Yaskawa INFORM job: A_ROOF_UPPER_0614_2_PAINT_1.JBI

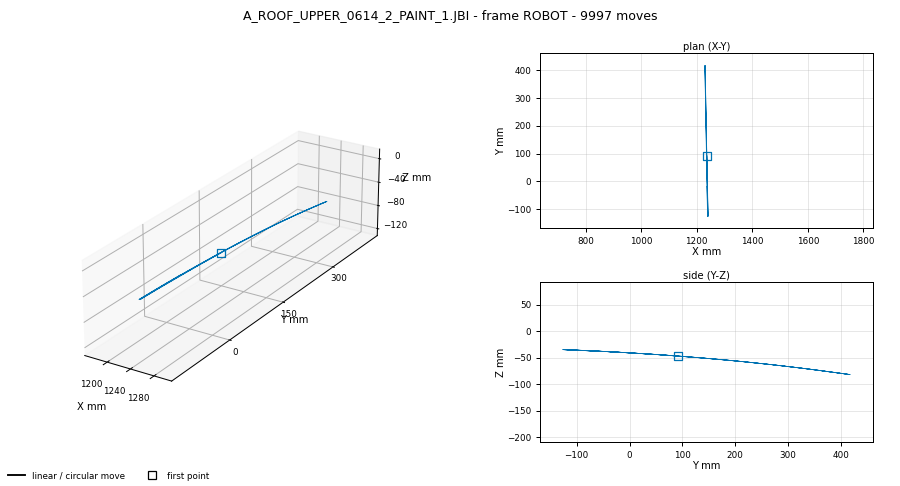
[picture p0: tool path of A_ROOF_UPPER_0614_2_PAINT_1.JBI in frame ROBOT, 9997 of 9997 moves have a stored position in this frame; points joined in program order, loops and branches not executed]
/JOB
//NAME A_ROOF_UPPER_0614_2_PAINT1
//POS
///NPOS 9997,0,0,0,0,0
///TOOL 1
///USER 0
///POSTYPE ROBOT
///RECTAN
///RCONF 1,0,0,0,0,0,0,0,0,0,0,0,0,0,0,0,0,0,0,0,0,0,0,0
C00000=1236.854,92.154,-46.600,-178.429,5.415,148.469
C00001=1236.860,91.904,-46.581,-178.431,5.414,148.469
C00002=1236.864,91.655,-46.563,-178.434,5.413,148.470
C00003=1236.868,91.406,-46.544,-178.436,5.413,148.471
C00004=1236.874,91.156,-46.525,-178.439,5.412,148.471
C00005=1236.879,90.907,-46.507,-178.441,5.411,148.472
C00006=1236.884,90.658,-46.489,-178.444,5.411,148.472
C00007=1236.888,90.409,-46.470,-178.446,5.410,148.473
C00008=1236.894,90.159,-46.452,-178.449,5.409,148.474
C00009=1236.898,89.911,-46.433,-178.452,5.409,148.474
C00010=1236.903,89.661,-46.415,-178.454,5.408,148.475
C00011=1236.907,89.411,-46.397,-178.456,5.407,148.476
C00012=1236.913,89.162,-46.378,-178.459,5.407,148.476
C00013=1236.918,88.913,-46.359,-178.462,5.406,148.477
C00014=1236.922,88.664,-46.341,-178.464,5.405,148.477
C00015=1236.927,88.414,-46.323,-178.467,5.404,148.478
C00016=1236.932,88.165,-46.305,-178.470,5.403,148.479
C00017=1236.937,87.916,-46.286,-178.472,5.402,148.479
C00018=1236.941,87.666,-46.268,-178.475,5.402,148.480
C00019=1236.946,87.417,-46.250,-178.477,5.401,148.480
C00020=1236.951,87.168,-46.232,-178.480,5.400,148.481
C00021=1236.956,86.919,-46.214,-178.482,5.400,148.482
C00022=1236.961,86.669,-46.195,-178.485,5.399,148.482
C00023=1236.966,86.420,-46.176,-178.487,5.398,148.483
C00024=1236.971,86.171,-46.158,-178.490,5.397,148.483
C00025=1236.976,85.922,-46.140,-178.492,5.397,148.484
C00026=1236.980,85.672,-46.122,-178.495,5.396,148.485
C00027=1236.985,85.423,-46.104,-178.497,5.396,148.485
C00028=1236.990,85.174,-46.086,-178.500,5.395,148.486
C00029=1236.995,84.924,-46.067,-178.502,5.394,148.486
C00030=1237.000,84.676,-46.048,-178.505,5.393,148.487
C00031=1237.004,84.426,-46.030,-178.507,5.393,148.488
C00032=1237.009,84.176,-46.012,-178.510,5.392,148.488
C00033=1237.014,83.927,-45.994,-178.513,5.392,148.489
C00034=1237.019,83.678,-45.976,-178.515,5.391,148.489
C00035=1237.024,83.429,-45.958,-178.517,5.390,148.490
C00036=1237.029,83.180,-45.940,-178.520,5.389,148.491
C00037=1237.033,82.930,-45.922,-178.523,5.389,148.491
C00038=1237.038,82.681,-45.904,-178.525,5.388,148.492
C00039=1237.043,82.432,-45.886,-178.527,5.387,148.492
C00040=1237.049,82.163,-45.866,-178.530,5.387,148.493
C00041=1237.054,81.895,-45.846,-178.533,5.386,148.494
C00042=1237.059,81.626,-45.827,-178.536,5.385,148.494
C00043=1237.064,81.358,-45.808,-178.539,5.384,148.495
C00044=1237.069,81.109,-45.790,-178.541,5.383,148.496
C00045=1237.074,80.860,-45.772,-178.544,5.383,148.496
C00046=1237.078,80.610,-45.753,-178.546,5.382,148.497
C00047=1237.083,80.361,-45.735,-178.549,5.382,148.498
C00048=1237.088,80.112,-45.717,-178.552,5.381,148.498
C00049=1237.093,79.862,-45.699,-178.554,5.380,148.499
C00050=1237.098,79.613,-45.682,-178.556,5.379,148.499
C00051=1237.103,79.364,-45.664,-178.559,5.379,148.500
C00052=1237.108,79.114,-45.646,-178.562,5.378,148.501
C00053=1237.113,78.865,-45.628,-178.564,5.378,148.501
C00054=1237.117,78.615,-45.610,-178.566,5.377,148.502
C00055=1237.122,78.366,-45.592,-178.569,5.376,148.502
C00056=1237.127,78.117,-45.574,-178.572,5.375,148.503
C00057=1237.132,77.868,-45.556,-178.574,5.375,148.504
C00058=1237.137,77.619,-45.538,-178.577,5.374,148.504
C00059=1237.142,77.369,-45.520,-178.580,5.374,148.505
C00060=1237.147,77.120,-45.503,-178.582,5.373,148.506
C00061=1237.152,76.870,-45.485,-178.584,5.372,148.506
C00062=1237.157,76.621,-45.467,-178.587,5.371,148.507
C00063=1237.162,76.372,-45.449,-178.590,5.371,148.508
C00064=1237.167,76.123,-45.431,-178.592,5.370,148.508
C00065=1237.172,75.873,-45.414,-178.595,5.370,148.509
C00066=1237.176,75.623,-45.395,-178.597,5.369,148.509
C00067=1237.180,75.374,-45.378,-178.600,5.368,148.510
C00068=1237.185,75.125,-45.360,-178.602,5.368,148.511
C00069=1237.190,74.876,-45.342,-178.605,5.367,148.511
C00070=1237.195,74.626,-45.325,-178.607,5.367,148.512
C00071=1237.200,74.377,-45.307,-178.610,5.367,148.513
C00072=1237.205,74.128,-45.289,-178.612,5.366,148.513
C00073=1237.210,73.879,-45.271,-178.614,5.365,148.514
C00074=1237.215,73.629,-45.253,-178.617,5.364,148.514
C00075=1237.220,73.380,-45.236,-178.620,5.364,148.515
C00076=1237.224,73.131,-45.218,-178.622,5.363,148.516
C00077=1237.230,72.881,-45.201,-178.625,5.363,148.516
C00078=1237.235,72.632,-45.183,-178.627,5.362,148.517
C00079=1237.240,72.383,-45.165,-178.630,5.361,148.517
C00080=1237.244,72.134,-45.147,-178.632,5.360,148.518
C00081=1237.249,71.884,-45.130,-178.635,5.360,148.519
C00082=1237.254,71.635,-45.112,-178.637,5.359,148.519
C00083=1237.259,71.386,-45.094,-178.640,5.359,148.520
C00084=1237.264,71.136,-45.077,-178.643,5.358,148.521
C00085=1237.269,70.887,-45.059,-178.645,5.357,148.521
C00086=1237.273,70.637,-45.042,-178.647,5.357,148.522
C00087=1237.278,70.388,-45.024,-178.650,5.356,148.522
C00088=1237.283,70.139,-45.006,-178.653,5.355,148.523
C00089=1237.288,69.889,-44.989,-178.655,5.355,148.524
C00090=1237.293,69.640,-44.972,-178.658,5.354,148.524
C00091=1237.298,69.390,-44.954,-178.661,5.354,148.525
C00092=1237.303,69.141,-44.936,-178.663,5.353,148.526
C00093=1237.308,68.892,-44.918,-178.666,5.352,148.526
C00094=1237.312,68.643,-44.902,-178.668,5.351,148.527
C00095=1237.317,68.393,-44.884,-178.670,5.352,148.528
C00096=1237.322,68.144,-44.866,-178.673,5.351,148.528
C00097=1237.327,67.894,-44.849,-178.675,5.350,148.529
C00098=1237.332,67.645,-44.832,-178.678,5.350,148.530
C00099=1237.337,67.396,-44.814,-178.681,5.349,148.530
C00100=1237.342,67.146,-44.797,-178.683,5.349,148.531
C00101=1237.346,66.897,-44.779,-178.685,5.348,148.531
C00102=1237.352,66.648,-44.762,-178.688,5.347,148.532
C00103=1237.357,66.399,-44.744,-178.691,5.347,148.533
C00104=1237.362,66.149,-44.727,-178.693,5.346,148.533
C00105=1237.366,65.900,-44.710,-178.696,5.345,148.534
C00106=1237.371,65.650,-44.692,-178.699,5.345,148.535
C00107=1237.376,65.401,-44.674,-178.701,5.344,148.535
C00108=1237.381,65.152,-44.658,-178.704,5.344,148.536
C00109=1237.386,64.903,-44.640,-178.706,5.343,148.536
C00110=1237.391,64.653,-44.623,-178.708,5.343,148.537
C00111=1237.395,64.403,-44.606,-178.711,5.342,148.538
C00112=1237.400,64.154,-44.588,-178.713,5.342,148.538
C00113=1237.405,63.905,-44.572,-178.716,5.341,148.539
C00114=1237.410,63.656,-44.554,-178.719,5.340,148.540
C00115=1237.415,63.406,-44.536,-178.721,5.340,148.540
C00116=1237.420,63.157,-44.520,-178.724,5.339,148.541
C00117=1237.425,62.908,-44.502,-178.726,5.339,148.542
C00118=1237.429,62.658,-44.485,-178.729,5.338,148.542
C00119=1237.434,62.409,-44.467,-178.731,5.337,148.543
C00120=1237.439,62.159,-44.450,-178.734,5.337,148.543
C00121=1237.444,61.910,-44.433,-178.736,5.336,148.544
C00122=1237.449,61.661,-44.415,-178.739,5.335,148.545
C00123=1237.454,61.412,-44.399,-178.741,5.336,148.545
C00124=1237.459,61.162,-44.382,-178.744,5.335,148.546
C00125=1237.464,60.912,-44.364,-178.746,5.334,148.547
C00126=1237.468,60.663,-44.347,-178.749,5.334,148.547
C00127=1237.474,60.414,-44.330,-178.752,5.333,148.548
C00128=1237.479,60.165,-44.313,-178.754,5.332,148.549
C00129=1237.484,59.916,-44.295,-178.756,5.332,148.549
C00130=1237.488,59.666,-44.279,-178.759,5.331,148.550
C00131=1237.493,59.416,-44.261,-178.762,5.331,148.551
C00132=1237.498,59.167,-44.245,-178.764,5.330,148.551
C00133=1237.503,58.918,-44.227,-178.767,5.329,148.552
C00134=1237.508,58.669,-44.210,-178.769,5.330,148.553
C00135=1237.513,58.419,-44.193,-178.772,5.329,148.553
C00136=1237.518,58.170,-44.177,-178.774,5.328,148.554
C00137=1237.523,57.920,-44.159,-178.777,5.328,148.555
C00138=1237.528,57.672,-44.142,-178.779,5.327,148.555
C00139=1237.533,57.422,-44.125,-178.782,5.326,148.556
C00140=1237.537,57.172,-44.108,-178.784,5.326,148.556
C00141=1237.542,56.923,-44.091,-178.787,5.325,148.557
C00142=1237.547,56.673,-44.074,-178.790,5.325,148.558
C00143=1237.553,56.424,-44.057,-178.792,5.325,148.558
C00144=1237.557,56.155,-44.039,-178.795,5.323,148.559
C00145=1237.563,55.887,-44.021,-178.798,5.323,148.560
C00146=1237.568,55.619,-44.003,-178.800,5.322,148.560
C00147=1237.573,55.350,-43.984,-178.803,5.322,148.561
C00148=1237.578,55.102,-43.967,-178.805,5.322,148.562
C00149=1237.583,54.852,-43.950,-178.808,5.321,148.562
C00150=1237.588,54.602,-43.933,-178.810,5.321,148.563
C00151=1237.592,54.353,-43.917,-178.813,5.320,148.564
C00152=1237.598,54.104,-43.900,-178.815,5.320,148.564
C00153=1237.603,53.854,-43.883,-178.818,5.319,148.565
C00154=1237.608,53.605,-43.866,-178.821,5.318,148.566
C00155=1237.612,53.355,-43.849,-178.823,5.318,148.566
C00156=1237.617,53.106,-43.833,-178.826,5.317,148.567
C00157=1237.623,52.856,-43.816,-178.828,5.317,148.568
C00158=1237.627,52.607,-43.799,-178.831,5.317,148.568
C00159=1237.633,52.358,-43.782,-178.833,5.316,148.569
C00160=1237.637,52.108,-43.765,-178.836,5.316,148.570
C00161=1237.642,51.859,-43.749,-178.838,5.315,148.570
C00162=1237.647,51.609,-43.731,-178.841,5.314,148.571
C00163=1237.652,51.360,-43.715,-178.843,5.314,148.571
C00164=1237.657,51.111,-43.698,-178.846,5.313,148.572
C00165=1237.662,50.861,-43.681,-178.848,5.313,148.573
C00166=1237.667,50.612,-43.665,-178.851,5.313,148.574
C00167=1237.672,50.363,-43.648,-178.853,5.312,148.574
C00168=1237.676,50.113,-43.632,-178.856,5.312,148.575
C00169=1237.682,49.864,-43.615,-178.859,5.311,148.576
C00170=1237.686,49.615,-43.598,-178.861,5.310,148.576
C00171=1237.691,49.365,-43.581,-178.864,5.310,148.577
C00172=1237.697,49.116,-43.564,-178.866,5.310,148.578
C00173=1237.701,48.867,-43.548,-178.869,5.309,148.578
C00174=1237.706,48.617,-43.531,-178.871,5.309,148.579
C00175=1237.712,48.367,-43.515,-178.874,5.308,148.580
C00176=1237.716,48.118,-43.498,-178.876,5.307,148.580
C00177=1237.721,47.868,-43.482,-178.879,5.307,148.581
C00178=1237.726,47.620,-43.465,-178.881,5.306,148.581
C00179=1237.731,47.370,-43.448,-178.883,5.306,148.582
C00180=1237.735,47.120,-43.431,-178.886,5.306,148.583
C00181=1237.740,46.872,-43.415,-178.889,5.305,148.583
C00182=1237.745,46.622,-43.399,-178.891,5.305,148.584
C00183=1237.750,46.372,-43.382,-178.894,5.304,148.585
C00184=1237.756,46.123,-43.365,-178.897,5.304,148.585
C00185=1237.760,45.873,-43.349,-178.899,5.303,148.586
C00186=1237.765,45.625,-43.333,-178.901,5.303,148.587
C00187=1237.770,45.375,-43.317,-178.904,5.303,148.587
C00188=1237.775,45.125,-43.299,-178.907,5.302,148.588
C00189=1237.780,44.876,-43.283,-178.909,5.301,148.589
C00190=1237.785,44.627,-43.266,-178.912,5.301,148.589
C00191=1237.790,44.378,-43.250,-178.914,5.300,148.590
C00192=1237.795,44.128,-43.234,-178.917,5.301,148.591
C00193=1237.799,43.878,-43.217,-178.919,5.300,148.591
C00194=1237.805,43.629,-43.200,-178.922,5.299,148.592
C00195=1237.810,43.379,-43.185,-178.924,5.299,148.593
C00196=1237.815,43.130,-43.168,-178.927,5.298,148.593
C00197=1237.819,42.881,-43.152,-178.929,5.297,148.594
C00198=1237.824,42.631,-43.135,-178.931,5.298,148.595
C00199=1237.829,42.382,-43.119,-178.934,5.297,148.595
C00200=1237.834,42.132,-43.102,-178.937,5.296,148.596
C00201=1237.839,41.883,-43.086,-178.939,5.296,148.597
C00202=1237.844,41.633,-43.070,-178.942,5.295,148.597
C00203=1237.849,41.384,-43.053,-178.944,5.295,148.598
C00204=1237.854,41.135,-43.037,-178.947,5.295,148.599
C00205=1237.859,40.885,-43.021,-178.949,5.294,148.599
C00206=1237.864,40.636,-43.005,-178.952,5.294,148.600
C00207=1237.868,40.387,-42.988,-178.954,5.293,148.601
C00208=1237.873,40.137,-42.972,-178.957,5.293,148.601
C00209=1237.878,39.888,-42.956,-178.960,5.292,148.602
C00210=1237.884,39.638,-42.939,-178.962,5.292,148.603
C00211=1237.889,39.388,-42.923,-178.964,5.292,148.603
C00212=1237.894,39.140,-42.906,-178.967,5.291,148.604
C00213=1237.898,38.890,-42.891,-178.970,5.291,148.605
C00214=1237.903,38.641,-42.874,-178.972,5.290,148.605
C00215=1237.908,38.391,-42.858,-178.974,5.290,148.606
C00216=1237.913,38.142,-42.842,-178.977,5.290,148.607
C00217=1237.918,37.892,-42.826,-178.980,5.289,148.607
C00218=1237.923,37.643,-42.810,-178.982,5.289,148.608
C00219=1237.928,37.393,-42.794,-178.985,5.288,148.609
C00220=1237.933,37.144,-42.777,-178.987,5.288,148.609
C00221=1237.938,36.895,-42.761,-178.990,5.288,148.610
C00222=1237.943,36.645,-42.745,-178.992,5.287,148.611
C00223=1237.947,36.396,-42.729,-178.995,5.287,148.611
C00224=1237.953,36.146,-42.713,-178.998,5.286,148.612
C00225=1237.957,35.897,-42.696,-179.000,5.285,148.613
C00226=1237.963,35.647,-42.681,-179.002,5.285,148.613
C00227=1237.967,35.397,-42.665,-179.005,5.285,148.614
C00228=1237.973,35.149,-42.648,-179.007,5.284,148.615
C00229=1237.978,34.899,-42.633,-179.010,5.284,148.615
C00230=1237.982,34.650,-42.616,-179.012,5.283,148.616
C00231=1237.988,34.400,-42.601,-179.014,5.283,148.617
C00232=1237.992,34.151,-42.584,-179.017,5.283,148.617
C00233=1237.998,33.901,-42.568,-179.020,5.282,148.618
C00234=1238.002,33.652,-42.552,-179.022,5.282,148.619
C00235=1238.008,33.402,-42.536,-179.025,5.281,148.619
C00236=1238.012,33.152,-42.520,-179.027,5.281,148.620
C00237=1238.017,32.904,-42.504,-179.030,5.281,148.621
C00238=1238.022,32.655,-42.489,-179.032,5.280,148.621
C00239=1238.027,32.404,-42.473,-179.035,5.280,148.622
C00240=1238.032,32.156,-42.457,-179.038,5.279,148.623
C00241=1238.037,31.906,-42.441,-179.040,5.279,148.623
C00242=1238.042,31.657,-42.424,-179.042,5.279,148.624
C00243=1238.047,31.407,-42.408,-179.045,5.278,148.625
C00244=1238.052,31.157,-42.393,-179.048,5.278,148.625
C00245=1238.057,30.908,-42.376,-179.050,5.278,148.626
C00246=1238.062,30.658,-42.360,-179.052,5.277,148.627
C00247=1238.066,30.409,-42.345,-179.055,5.277,148.627
C00248=1238.072,30.141,-42.328,-179.058,5.276,148.628
C00249=1238.077,29.872,-42.311,-179.061,5.276,148.629
C00250=1238.083,29.603,-42.294,-179.064,5.275,148.630
C00251=1238.088,29.335,-42.277,-179.066,5.275,148.630
C00252=1238.093,29.086,-42.261,-179.068,5.275,148.631
C00253=1238.098,28.836,-42.245,-179.071,5.275,148.632
C00254=1238.103,28.587,-42.230,-179.074,5.274,148.632
C00255=1238.108,28.337,-42.214,-179.076,5.273,148.633
C00256=1238.112,28.088,-42.198,-179.079,5.273,148.634
C00257=1238.118,27.838,-42.182,-179.081,5.273,148.635
C00258=1238.123,27.588,-42.166,-179.084,5.273,148.635
C00259=1238.128,27.339,-42.150,-179.086,5.272,148.636
C00260=1238.133,27.090,-42.135,-179.089,5.271,148.637
C00261=1238.137,26.840,-42.119,-179.091,5.272,148.637
C00262=1238.143,26.591,-42.103,-179.094,5.271,148.638
C00263=1238.148,26.341,-42.088,-179.096,5.271,148.639
C00264=1238.152,26.092,-42.072,-179.099,5.270,148.639
C00265=1238.157,25.842,-42.057,-179.101,5.269,148.640
C00266=1238.163,25.593,-42.041,-179.104,5.270,148.641
C00267=1238.167,25.343,-42.024,-179.106,5.269,148.641
C00268=1238.172,25.094,-42.009,-179.109,5.269,148.642
C00269=1238.177,24.845,-41.994,-179.111,5.268,148.643
C00270=1238.182,24.595,-41.978,-179.114,5.268,148.643
C00271=1238.187,24.345,-41.962,-179.116,5.268,148.644
C00272=1238.192,24.096,-41.947,-179.119,5.267,148.645
C00273=1238.198,23.847,-41.932,-179.121,5.267,148.645
C00274=1238.202,23.597,-41.916,-179.124,5.267,148.646
C00275=1238.207,23.348,-41.899,-179.126,5.266,148.647
C00276=1238.212,23.099,-41.884,-179.129,5.266,148.647
C00277=1238.217,22.849,-41.868,-179.131,5.265,148.648
C00278=1238.222,22.599,-41.853,-179.134,5.265,148.649
C00279=1238.227,22.350,-41.838,-179.136,5.265,148.649
C00280=1238.232,22.101,-41.822,-179.139,5.264,148.650
C00281=1238.237,21.851,-41.806,-179.142,5.264,148.651
C00282=1238.242,21.602,-41.791,-179.144,5.264,148.652
C00283=1238.247,21.352,-41.776,-179.146,5.264,148.652
C00284=1238.252,21.102,-41.760,-179.149,5.263,148.653
C00285=1238.256,20.853,-41.745,-179.152,5.262,148.654
C00286=1238.262,20.604,-41.729,-179.154,5.263,148.654
C00287=1238.267,20.354,-41.714,-179.156,5.262,148.655
C00288=1238.271,20.105,-41.698,-179.159,5.262,148.656
C00289=1238.277,19.855,-41.683,-179.162,5.261,148.656
C00290=1238.282,19.606,-41.667,-179.164,5.261,148.657
C00291=1238.287,19.357,-41.652,-179.166,5.261,148.658
C00292=1238.292,19.107,-41.637,-179.169,5.260,148.658
C00293=1238.296,18.857,-41.621,-179.172,5.260,148.659
C00294=1238.302,18.608,-41.606,-179.174,5.260,148.660
C00295=1238.307,18.359,-41.590,-179.177,5.260,148.661
C00296=1238.312,18.110,-41.575,-179.179,5.259,148.661
C00297=1238.317,17.859,-41.560,-179.182,5.259,148.662
C00298=1238.321,17.610,-41.545,-179.184,5.259,148.663
C00299=1238.327,17.360,-41.529,-179.187,5.258,148.663
C00300=1238.331,17.111,-41.514,-179.189,5.258,148.664
C00301=1238.337,16.862,-41.499,-179.192,5.257,148.665
C00302=1238.342,16.612,-41.483,-179.194,5.257,148.665
C00303=1238.346,16.363,-41.468,-179.197,5.257,148.666
C00304=1238.352,16.113,-41.452,-179.199,5.256,148.667
C00305=1238.357,15.864,-41.438,-179.202,5.257,148.667
C00306=1238.362,15.614,-41.422,-179.204,5.256,148.668
C00307=1238.366,15.364,-41.407,-179.207,5.256,148.669
C00308=1238.371,15.115,-41.391,-179.209,5.255,148.670
C00309=1238.376,14.866,-41.376,-179.212,5.255,148.670
C00310=1238.381,14.616,-41.361,-179.214,5.255,148.671
C00311=1238.386,14.367,-41.346,-179.217,5.254,148.672
C00312=1238.392,14.117,-41.331,-179.219,5.254,148.672
C00313=1238.396,13.868,-41.316,-179.222,5.254,148.673
C00314=1238.401,13.618,-41.300,-179.224,5.253,148.674
C00315=1238.406,13.369,-41.285,-179.227,5.253,148.674
C00316=1238.412,13.119,-41.270,-179.229,5.253,148.675
C00317=1238.416,12.870,-41.255,-179.232,5.252,148.676
C00318=1238.422,12.621,-41.239,-179.234,5.252,148.676
C00319=1238.426,12.371,-41.224,-179.237,5.251,148.677
C00320=1238.432,12.121,-41.210,-179.239,5.252,148.678
C00321=1238.436,11.872,-41.194,-179.242,5.251,148.678
C00322=1238.441,11.622,-41.179,-179.244,5.251,148.679
C00323=1238.446,11.372,-41.164,-179.246,5.251,148.680
C00324=1238.452,11.123,-41.149,-179.249,5.250,148.680
C00325=1238.456,10.874,-41.134,-179.252,5.250,148.681
C00326=1238.461,10.625,-41.119,-179.255,5.250,148.682
C00327=1238.467,10.375,-41.104,-179.257,5.250,148.683
C00328=1238.471,10.126,-41.089,-179.260,5.249,148.683
C00329=1238.476,9.876,-41.073,-179.262,5.249,148.684
C00330=1238.481,9.626,-41.059,-179.264,5.249,148.685
C00331=1238.486,9.377,-41.044,-179.267,5.248,148.686
C00332=1238.491,9.127,-41.029,-179.270,5.248,148.686
C00333=1238.496,8.878,-41.014,-179.272,5.247,148.687
C00334=1238.501,8.628,-40.998,-179.274,5.248,148.688
C00335=1238.506,8.379,-40.984,-179.277,5.247,148.688
C00336=1238.511,8.130,-40.969,-179.280,5.247,148.689
C00337=1238.516,7.880,-40.953,-179.282,5.247,148.690
C00338=1238.521,7.630,-40.939,-179.284,5.246,148.690
C00339=1238.526,7.381,-40.924,-179.287,5.246,148.691
C00340=1238.532,7.131,-40.909,-179.289,5.246,148.692
C00341=1238.536,6.882,-40.894,-179.292,5.245,148.692
C00342=1238.542,6.632,-40.879,-179.294,5.245,148.693
C00343=1238.546,6.382,-40.864,-179.297,5.244,148.694
C00344=1238.551,6.133,-40.849,-179.299,5.245,148.694
C00345=1238.556,5.883,-40.834,-179.302,5.244,148.695
C00346=1238.561,5.634,-40.819,-179.304,5.244,148.696
C00347=1238.566,5.385,-40.805,-179.307,5.244,148.697
C00348=1238.571,5.135,-40.790,-179.310,5.244,148.697
C00349=1238.576,4.885,-40.775,-179.312,5.243,148.698
C00350=1238.581,4.636,-40.760,-179.314,5.243,148.699
C00351=1238.586,4.387,-40.746,-179.317,5.243,148.700
C00352=1238.592,4.118,-40.729,-179.320,5.242,148.700
C00353=1238.597,3.849,-40.714,-179.322,5.242,148.701
C00354=1238.602,3.580,-40.698,-179.325,5.242,148.702
C00355=1238.608,3.311,-40.682,-179.328,5.242,148.702
C00356=1238.613,3.062,-40.667,-179.330,5.241,148.703
C00357=1238.618,2.812,-40.652,-179.333,5.241,148.704
C00358=1238.623,2.563,-40.637,-179.335,5.241,148.705
C00359=1238.628,2.313,-40.623,-179.338,5.241,148.705
C00360=1238.633,2.064,-40.608,-179.340,5.240,148.706
C00361=1238.638,1.814,-40.593,-179.343,5.239,148.707
C00362=1238.642,1.564,-40.579,-179.345,5.240,148.707
C00363=1238.648,1.315,-40.563,-179.348,5.239,148.708
C00364=1238.653,1.065,-40.549,-179.350,5.239,148.709
C00365=1238.657,0.816,-40.534,-179.352,5.239,148.709
C00366=1238.663,0.567,-40.520,-179.355,5.238,148.710
C00367=1238.669,0.317,-40.505,-179.358,5.238,148.711
C00368=1238.673,0.068,-40.490,-179.360,5.238,148.712
C00369=1238.678,-0.182,-40.476,-179.363,5.238,148.712
C00370=1238.683,-0.431,-40.462,-179.365,5.237,148.713
C00371=1238.688,-0.680,-40.447,-179.368,5.238,148.714
C00372=1238.694,-0.930,-40.432,-179.370,5.237,148.714
C00373=1238.699,-1.180,-40.418,-179.373,5.237,148.715
C00374=1238.703,-1.429,-40.403,-179.375,5.237,148.716
C00375=1238.708,-1.679,-40.388,-179.378,5.236,148.716
C00376=1238.713,-1.929,-40.374,-179.380,5.236,148.717
C00377=1238.718,-2.178,-40.359,-179.382,5.236,148.718
C00378=1238.723,-2.427,-40.345,-179.385,5.236,148.719
C00379=1238.728,-2.678,-40.330,-179.388,5.235,148.719
C00380=1238.733,-2.927,-40.316,-179.390,5.235,148.720
C00381=1238.738,-3.176,-40.301,-179.392,5.235,148.721
C00382=1238.744,-3.425,-40.287,-179.395,5.234,148.721
C00383=1238.749,-3.675,-40.273,-179.398,5.235,148.722
C00384=1238.753,-3.925,-40.258,-179.400,5.234,148.723
C00385=1238.758,-4.174,-40.243,-179.403,5.234,148.724
C00386=1238.763,-4.424,-40.229,-179.405,5.234,148.724
C00387=1238.769,-4.674,-40.214,-179.408,5.234,148.725
C00388=1238.774,-4.923,-40.200,-179.410,5.233,148.726
C00389=1238.778,-5.172,-40.185,-179.412,5.233,148.726
C00390=1238.783,-5.422,-40.171,-179.415,5.233,148.727
C00391=1238.788,-5.672,-40.156,-179.418,5.232,148.728
C00392=1238.794,-5.921,-40.142,-179.420,5.233,148.728
C00393=1238.799,-6.170,-40.128,-179.422,5.232,148.729
C00394=1238.804,-6.420,-40.114,-179.425,5.231,148.730
C00395=1238.808,-6.669,-40.099,-179.427,5.232,148.731
C00396=1238.813,-6.919,-40.085,-179.430,5.231,148.731
C00397=1238.818,-7.169,-40.070,-179.432,5.231,148.732
C00398=1238.823,-7.418,-40.056,-179.435,5.231,148.733
C00399=1238.829,-7.667,-40.042,-179.438,5.231,148.734
C00400=1238.834,-7.917,-40.028,-179.440,5.230,148.734
C00401=1238.839,-8.167,-40.014,-179.442,5.231,148.735
C00402=1238.844,-8.417,-39.999,-179.445,5.230,148.736
C00403=1238.848,-8.666,-39.984,-179.447,5.230,148.736
C00404=1238.853,-8.915,-39.970,-179.450,5.230,148.737
C00405=1238.858,-9.165,-39.956,-179.452,5.229,148.738
C00406=1238.864,-9.414,-39.942,-179.455,5.230,148.738
C00407=1238.869,-9.664,-39.928,-179.457,5.229,148.739
C00408=1238.874,-9.914,-39.913,-179.460,5.228,148.740
C00409=1238.879,-10.163,-39.899,-179.462,5.229,148.740
C00410=1238.884,-10.413,-39.885,-179.465,5.228,148.741
C00411=1238.889,-10.662,-39.871,-179.467,5.228,148.742
C00412=1238.894,-10.912,-39.857,-179.470,5.228,148.743
C00413=1238.899,-11.161,-39.842,-179.473,5.228,148.743
C00414=1238.904,-11.411,-39.828,-179.475,5.227,148.744
C00415=1238.909,-11.661,-39.814,-179.477,5.228,148.745
C00416=1238.915,-11.910,-39.800,-179.480,5.227,148.746
C00417=1238.920,-12.160,-39.785,-179.482,5.227,148.746
C00418=1238.924,-12.409,-39.771,-179.485,5.227,148.747
C00419=1238.929,-12.659,-39.757,-179.487,5.226,148.748
C00420=1238.934,-12.909,-39.743,-179.489,5.227,148.748
C00421=1238.940,-13.158,-39.729,-179.492,5.226,148.749
C00422=1238.944,-13.407,-39.715,-179.495,5.226,148.750
C00423=1238.949,-13.657,-39.701,-179.497,5.226,148.750
C00424=1238.954,-13.906,-39.687,-179.499,5.225,148.751
C00425=1238.960,-14.155,-39.673,-179.503,5.225,148.752
C00426=1238.965,-14.405,-39.658,-179.505,5.225,148.753
C00427=1238.970,-14.655,-39.644,-179.507,5.225,148.753
C00428=1238.974,-14.905,-39.630,-179.509,5.225,148.754
C00429=1238.980,-15.154,-39.617,-179.512,5.225,148.755
C00430=1238.985,-15.404,-39.602,-179.515,5.224,148.755
C00431=1238.990,-15.653,-39.589,-179.517,5.224,148.756
C00432=1238.994,-15.903,-39.574,-179.519,5.224,148.757
C00433=1239.000,-16.152,-39.560,-179.522,5.223,148.758
C00434=1239.005,-16.402,-39.546,-179.524,5.224,148.758
C00435=1239.010,-16.651,-39.532,-179.527,5.223,148.759
C00436=1239.015,-16.901,-39.518,-179.529,5.223,148.760
C00437=1239.020,-17.151,-39.505,-179.532,5.223,148.761
C00438=1239.025,-17.400,-39.491,-179.535,5.223,148.761
C00439=1239.030,-17.650,-39.476,-179.537,5.223,148.762
C00440=1239.035,-17.899,-39.463,-179.539,5.223,148.763
C00441=1239.040,-18.149,-39.448,-179.542,5.222,148.763
C00442=1239.046,-18.399,-39.435,-179.544,5.222,148.764
C00443=1239.051,-18.648,-39.421,-179.547,5.222,148.765
C00444=1239.055,-18.897,-39.407,-179.549,5.222,148.765
C00445=1239.060,-19.147,-39.393,-179.552,5.222,148.766
C00446=1239.065,-19.397,-39.379,-179.554,5.221,148.767
C00447=1239.071,-19.646,-39.365,-179.556,5.221,148.768
C00448=1239.075,-19.896,-39.352,-179.559,5.221,148.768
C00449=1239.080,-20.146,-39.337,-179.562,5.220,148.769
C00450=1239.086,-20.395,-39.323,-179.564,5.221,148.770
C00451=1239.091,-20.645,-39.310,-179.567,5.220,148.771
C00452=1239.095,-20.894,-39.296,-179.569,5.221,148.771
C00453=1239.101,-21.143,-39.282,-179.572,5.220,148.772
C00454=1239.106,-21.393,-39.268,-179.574,5.220,148.773
C00455=1239.111,-21.643,-39.254,-179.576,5.220,148.773
C00456=1239.117,-21.912,-39.240,-179.579,5.219,148.774
C00457=1239.122,-22.181,-39.225,-179.582,5.219,148.775
C00458=1239.127,-22.451,-39.210,-179.584,5.220,148.776
C00459=1239.133,-22.720,-39.195,-179.587,5.219,148.776
C00460=1239.138,-22.969,-39.182,-179.590,5.219,148.777
C00461=1239.143,-23.218,-39.168,-179.592,5.219,148.778
C00462=1239.148,-23.469,-39.154,-179.595,5.219,148.779
C00463=1239.153,-23.718,-39.140,-179.598,5.218,148.779
C00464=1239.158,-23.967,-39.127,-179.600,5.219,148.780
C00465=1239.163,-24.217,-39.114,-179.602,5.218,148.781
C00466=1239.168,-24.466,-39.099,-179.604,5.218,148.781
C00467=1239.173,-24.717,-39.086,-179.607,5.218,148.782
C00468=1239.179,-24.966,-39.072,-179.610,5.217,148.783
C00469=1239.183,-25.215,-39.058,-179.612,5.218,148.784
C00470=1239.188,-25.465,-39.045,-179.614,5.217,148.784
C00471=1239.194,-25.714,-39.031,-179.617,5.217,148.785
C00472=1239.199,-25.965,-39.018,-179.619,5.217,148.786
C00473=1239.204,-26.213,-39.004,-179.622,5.217,148.787
C00474=1239.209,-26.463,-38.990,-179.624,5.217,148.787
C00475=1239.214,-26.713,-38.977,-179.627,5.216,148.788
C00476=1239.219,-26.962,-38.963,-179.629,5.217,148.789
C00477=1239.224,-27.212,-38.950,-179.632,5.216,148.789
C00478=1239.229,-27.461,-38.936,-179.634,5.216,148.790
C00479=1239.234,-27.711,-38.923,-179.637,5.216,148.791
C00480=1239.240,-27.960,-38.909,-179.639,5.216,148.791
C00481=1239.244,-28.210,-38.896,-179.641,5.216,148.792
C00482=1239.249,-28.460,-38.882,-179.644,5.215,148.793
C00483=1239.254,-28.709,-38.869,-179.647,5.215,148.794
C00484=1239.259,-28.959,-38.855,-179.649,5.215,148.794
C00485=1239.265,-29.209,-38.842,-179.652,5.215,148.795
C00486=1239.269,-29.458,-38.828,-179.654,5.215,148.796
C00487=1239.275,-29.708,-38.815,-179.657,5.215,148.797
C00488=1239.279,-29.957,-38.801,-179.659,5.214,148.797
C00489=1239.285,-30.207,-38.788,-179.661,5.215,148.798
C00490=1239.289,-30.456,-38.774,-179.664,5.214,148.799
C00491=1239.295,-30.706,-38.761,-179.666,5.214,148.799
C00492=1239.300,-30.956,-38.748,-179.669,5.214,148.800
C00493=1239.305,-31.205,-38.734,-179.671,5.214,148.801
C00494=1239.311,-31.455,-38.720,-179.674,5.214,148.801
C00495=1239.315,-31.705,-38.707,-179.676,5.213,148.802
C00496=1239.321,-31.954,-38.694,-179.679,5.214,148.803
C00497=1239.325,-32.204,-38.680,-179.681,5.213,148.804
C00498=1239.331,-32.453,-38.667,-179.683,5.214,148.804
C00499=1239.335,-32.703,-38.654,-179.686,5.213,148.805
C00500=1239.341,-32.952,-38.640,-179.689,5.213,148.806
C00501=1239.345,-33.202,-38.627,-179.691,5.213,148.807
C00502=1239.351,-33.452,-38.614,-179.694,5.212,148.807
C00503=1239.355,-33.701,-38.600,-179.696,5.213,148.808
C00504=1239.361,-33.951,-38.587,-179.698,5.212,148.809
C00505=1239.366,-34.200,-38.574,-179.700,5.212,148.809
C00506=1239.371,-34.450,-38.560,-179.703,5.212,148.810
C00507=1239.376,-34.699,-38.547,-179.706,5.212,148.811
C00508=1239.381,-34.949,-38.534,-179.708,5.212,148.812
C00509=1239.387,-35.198,-38.520,-179.711,5.212,148.812
C00510=1239.391,-35.448,-38.507,-179.713,5.212,148.813
C00511=1239.397,-35.698,-38.494,-179.716,5.211,148.814
C00512=1239.401,-35.947,-38.481,-179.718,5.212,148.814
C00513=1239.407,-36.197,-38.467,-179.720,5.211,148.815
C00514=1239.412,-36.447,-38.454,-179.723,5.211,148.816
C00515=1239.417,-36.696,-38.442,-179.725,5.211,148.817
C00516=1239.422,-36.946,-38.428,-179.728,5.210,148.817
C00517=1239.427,-37.195,-38.415,-179.730,5.211,148.818
C00518=1239.433,-37.445,-38.402,-179.733,5.211,148.819
C00519=1239.437,-37.695,-38.389,-179.735,5.211,148.820
C00520=1239.443,-37.944,-38.375,-179.738,5.210,148.820
C00521=1239.447,-38.194,-38.362,-179.741,5.210,148.821
C00522=1239.452,-38.443,-38.349,-179.743,5.210,148.822
C00523=1239.458,-38.694,-38.336,-179.745,5.210,148.822
C00524=1239.463,-38.943,-38.323,-179.747,5.210,148.823
C00525=1239.467,-39.192,-38.310,-179.750,5.210,148.824
C00526=1239.473,-39.442,-38.296,-179.752,5.210,148.825
C00527=1239.478,-39.691,-38.284,-179.755,5.209,148.825
C00528=1239.482,-39.941,-38.271,-179.757,5.209,148.826
C00529=1239.488,-40.191,-38.257,-179.760,5.210,148.827
C00530=1239.493,-40.440,-38.245,-179.763,5.209,148.828
C00531=1239.498,-40.690,-38.231,-179.765,5.209,148.828
C00532=1239.503,-40.939,-38.218,-179.767,5.209,148.829
C00533=1239.508,-41.189,-38.205,-179.770,5.209,148.830
C00534=1239.513,-41.439,-38.192,-179.772,5.209,148.830
C00535=1239.519,-41.688,-38.179,-179.775,5.208,148.831
C00536=1239.524,-41.938,-38.166,-179.777,5.208,148.832
C00537=1239.529,-42.188,-38.154,-179.780,5.208,148.832
C00538=1239.534,-42.437,-38.140,-179.782,5.208,148.833
C00539=1239.539,-42.687,-38.127,-179.784,5.208,148.834
C00540=1239.544,-42.936,-38.114,-179.787,5.208,148.835
C00541=1239.549,-43.186,-38.101,-179.790,5.208,148.836
C00542=1239.554,-43.436,-38.088,-179.792,5.208,148.836
C00543=1239.559,-43.685,-38.075,-179.794,5.208,148.837
C00544=1239.564,-43.935,-38.062,-179.797,5.207,148.838
C00545=1239.570,-44.185,-38.049,-179.799,5.208,148.838
C00546=1239.575,-44.434,-38.037,-179.802,5.207,148.839
C00547=1239.579,-44.684,-38.024,-179.804,5.207,148.840
C00548=1239.584,-44.933,-38.011,-179.807,5.207,148.840
C00549=1239.590,-45.183,-37.998,-179.809,5.207,148.841
C00550=1239.595,-45.433,-37.985,-179.812,5.207,148.842
C00551=1239.600,-45.682,-37.972,-179.814,5.207,148.843
C00552=1239.605,-45.932,-37.960,-179.817,5.207,148.843
C00553=1239.610,-46.182,-37.946,-179.819,5.206,148.844
C00554=1239.616,-46.431,-37.934,-179.821,5.207,148.845
C00555=1239.621,-46.681,-37.921,-179.824,5.206,148.846
C00556=1239.625,-46.931,-37.908,-179.826,5.206,148.846
C00557=1239.630,-47.180,-37.895,-179.829,5.206,148.847
C00558=1239.636,-47.429,-37.882,-179.831,5.206,148.848
C00559=1239.641,-47.679,-37.870,-179.833,5.206,148.848
C00560=1239.646,-47.949,-37.856,-179.836,5.206,148.849
C00561=1239.652,-48.219,-37.842,-179.839,5.206,148.850
C00562=1239.658,-48.488,-37.828,-179.841,5.206,148.851
C00563=1239.663,-48.757,-37.815,-179.844,5.206,148.852
C00564=1239.668,-49.007,-37.801,-179.847,5.206,148.852
C00565=1239.673,-49.258,-37.789,-179.849,5.205,148.853
C00566=1239.678,-49.507,-37.777,-179.851,5.206,148.854
C00567=1239.684,-49.756,-37.764,-179.854,5.205,148.854
C00568=1239.689,-50.006,-37.751,-179.856,5.205,148.855
C00569=1239.693,-50.256,-37.738,-179.859,5.205,148.856
C00570=1239.698,-50.505,-37.726,-179.861,5.205,148.857
C00571=1239.704,-50.755,-37.713,-179.864,5.205,148.857
C00572=1239.709,-51.005,-37.700,-179.866,5.205,148.858
C00573=1239.714,-51.254,-37.688,-179.869,5.205,148.859
C00574=1239.719,-51.504,-37.675,-179.871,5.205,148.860
C00575=1239.724,-51.753,-37.663,-179.874,5.205,148.860
C00576=1239.729,-52.003,-37.650,-179.876,5.205,148.861
C00577=1239.734,-52.252,-37.637,-179.878,5.205,148.862
C00578=1239.739,-52.502,-37.625,-179.881,5.204,148.862
C00579=1239.745,-52.752,-37.613,-179.883,5.204,148.863
C00580=1239.750,-53.001,-37.600,-179.886,5.204,148.864
C00581=1239.755,-53.251,-37.586,-179.888,5.204,148.865
C00582=1239.760,-53.501,-37.574,-179.890,5.204,148.865
C00583=1239.766,-53.751,-37.562,-179.893,5.204,148.866
C00584=1239.771,-54.000,-37.549,-179.896,5.204,148.867
C00585=1239.775,-54.250,-37.536,-179.898,5.204,148.868
C00586=1239.780,-54.499,-37.524,-179.900,5.204,148.868
C00587=1239.786,-54.749,-37.512,-179.903,5.204,148.869
C00588=1239.791,-54.998,-37.499,-179.905,5.204,148.870
C00589=1239.796,-55.248,-37.487,-179.907,5.204,148.870
C00590=1239.800,-55.498,-37.474,-179.910,5.203,148.871
C00591=1239.806,-55.748,-37.462,-179.912,5.204,148.872
C00592=1239.811,-55.997,-37.449,-179.915,5.203,148.873
C00593=1239.816,-56.246,-37.437,-179.917,5.203,148.873
C00594=1239.822,-56.496,-37.425,-179.919,5.203,148.874
C00595=1239.826,-56.746,-37.412,-179.922,5.203,148.875
C00596=1239.831,-56.996,-37.399,-179.925,5.203,148.876
C00597=1239.837,-57.246,-37.387,-179.927,5.203,148.876
C00598=1239.842,-57.495,-37.375,-179.929,5.203,148.877
C00599=1239.847,-57.744,-37.362,-179.932,5.203,148.878
C00600=1239.852,-57.994,-37.350,-179.934,5.203,148.878
C00601=1239.857,-58.244,-37.337,-179.937,5.202,148.879
C00602=1239.862,-58.494,-37.325,-179.939,5.203,148.880
C00603=1239.867,-58.743,-37.313,-179.942,5.202,148.880
C00604=1239.873,-58.993,-37.300,-179.944,5.203,148.881
C00605=1239.878,-59.242,-37.288,-179.946,5.202,148.882
C00606=1239.883,-59.492,-37.276,-179.949,5.202,148.883
C00607=1239.888,-59.741,-37.263,-179.952,5.202,148.884
C00608=1239.893,-59.992,-37.251,-179.954,5.203,148.884
C00609=1239.897,-60.241,-37.239,-179.956,5.202,148.885
C00610=1239.903,-60.490,-37.226,-179.959,5.202,148.886
C00611=1239.908,-60.740,-37.214,-179.961,5.202,148.886
C00612=1239.913,-60.990,-37.202,-179.963,5.202,148.887
C00613=1239.919,-61.240,-37.190,-179.966,5.202,148.888
C00614=1239.924,-61.489,-37.177,-179.969,5.201,148.888
C00615=1239.929,-61.739,-37.165,-179.971,5.202,148.889
C00616=1239.934,-61.989,-37.152,-179.973,5.201,148.890
C00617=1239.939,-62.239,-37.140,-179.975,5.201,148.891
C00618=1239.944,-62.488,-37.128,-179.978,5.201,148.891
C00619=1239.949,-62.738,-37.117,-179.980,5.201,148.892
C00620=1239.954,-62.987,-37.104,-179.983,5.201,148.893
C00621=1239.959,-63.237,-37.092,-179.985,5.202,148.894
C00622=1239.965,-63.486,-37.079,-179.988,5.201,148.894
C00623=1239.970,-63.736,-37.068,-179.990,5.201,148.895
C00624=1239.975,-63.985,-37.055,-179.993,5.201,148.896
C00625=1239.981,-64.235,-37.043,-179.995,5.201,148.896
C00626=1239.986,-64.485,-37.031,-179.998,5.201,148.897
C00627=1239.990,-64.734,-37.019,-180.000,5.201,148.898
C00628=1239.995,-64.984,-37.006,179.998,5.201,148.899
C00629=1240.000,-65.234,-36.994,179.995,5.201,148.899
C00630=1240.005,-65.484,-36.982,179.993,5.200,148.900
C00631=1240.011,-65.734,-36.970,179.991,5.201,148.901
C00632=1240.016,-65.983,-36.959,179.988,5.201,148.902
C00633=1240.021,-66.233,-36.946,179.985,5.201,148.902
C00634=1240.026,-66.482,-36.934,179.983,5.200,148.903
C00635=1240.031,-66.732,-36.922,179.981,5.201,148.904
C00636=1240.037,-66.982,-36.910,179.978,5.200,148.904
C00637=1240.042,-67.232,-36.898,179.976,5.201,148.905
C00638=1240.046,-67.481,-36.886,179.973,5.200,148.906
C00639=1240.052,-67.731,-36.874,179.971,5.201,148.907
C00640=1240.057,-67.980,-36.861,179.969,5.200,148.907
C00641=1240.062,-68.230,-36.849,179.966,5.200,148.908
C00642=1240.067,-68.479,-36.838,179.964,5.200,148.909
C00643=1240.072,-68.729,-36.825,179.962,5.200,148.909
C00644=1240.078,-68.979,-36.814,179.959,5.200,148.910
C00645=1240.083,-69.229,-36.802,179.956,5.200,148.911
C00646=1240.088,-69.478,-36.790,179.954,5.200,148.912
C00647=1240.093,-69.728,-36.778,179.952,5.200,148.913
C00648=1240.098,-69.978,-36.766,179.949,5.200,148.913
C00649=1240.103,-70.227,-36.753,179.947,5.200,148.914
C00650=1240.108,-70.476,-36.742,179.944,5.200,148.915
C00651=1240.114,-70.726,-36.730,179.942,5.200,148.915
C00652=1240.119,-70.976,-36.718,179.939,5.200,148.916
C00653=1240.124,-71.226,-36.706,179.937,5.200,148.917
C00654=1240.129,-71.475,-36.694,179.935,5.199,148.917
C00655=1240.134,-71.725,-36.682,179.933,5.200,148.918
C00656=1240.140,-71.975,-36.671,179.930,5.199,148.919
C00657=1240.144,-72.224,-36.659,179.928,5.200,148.920
C00658=1240.150,-72.474,-36.647,179.925,5.199,148.920
C00659=1240.155,-72.724,-36.635,179.923,5.200,148.921
C00660=1240.160,-72.974,-36.624,179.920,5.199,148.922
C00661=1240.165,-73.223,-36.611,179.918,5.200,148.923
C00662=1240.170,-73.473,-36.599,179.915,5.199,148.923
C00663=1240.175,-73.723,-36.588,179.913,5.200,148.924
C00664=1240.181,-73.992,-36.575,179.910,5.199,148.925
C00665=1240.186,-74.263,-36.562,179.908,5.199,148.925
C00666=1240.193,-74.533,-36.549,179.905,5.199,148.926
C00667=1240.198,-74.803,-36.536,179.902,5.199,148.927
C00668=1240.203,-75.052,-36.525,179.900,5.199,148.928
C00669=1240.208,-75.302,-36.513,179.898,5.199,148.929
C00670=1240.213,-75.552,-36.502,179.896,5.199,148.929
C00671=1240.218,-75.802,-36.490,179.893,5.199,148.930
C00672=1240.224,-76.052,-36.478,179.891,5.199,148.931
C00673=1240.228,-76.302,-36.467,179.888,5.198,148.931
C00674=1240.234,-76.551,-36.454,179.886,5.199,148.932
C00675=1240.240,-76.800,-36.442,179.883,5.199,148.933
C00676=1240.244,-77.050,-36.431,179.881,5.199,148.934
C00677=1240.250,-77.300,-36.419,179.878,5.198,148.934
C00678=1240.254,-77.549,-36.408,179.876,5.199,148.935
C00679=1240.260,-77.799,-36.396,179.873,5.198,148.936
C00680=1240.265,-78.049,-36.385,179.871,5.199,148.937
C00681=1240.270,-78.299,-36.373,179.869,5.198,148.937
C00682=1240.275,-78.549,-36.361,179.867,5.199,148.938
C00683=1240.280,-78.798,-36.350,179.864,5.198,148.939
C00684=1240.286,-79.048,-36.338,179.862,5.198,148.939
C00685=1240.291,-79.297,-36.327,179.859,5.198,148.940
C00686=1240.296,-79.547,-36.315,179.857,5.198,148.941
C00687=1240.301,-79.796,-36.303,179.854,5.198,148.942
C00688=1240.306,-80.046,-36.291,179.852,5.198,148.942
C00689=1240.311,-80.296,-36.280,179.850,5.198,148.943
C00690=1240.316,-80.546,-36.268,179.847,5.198,148.944
C00691=1240.321,-80.795,-36.257,179.844,5.198,148.945
C00692=1240.327,-81.045,-36.245,179.842,5.198,148.945
C00693=1240.332,-81.294,-36.234,179.840,5.199,148.946
C00694=1240.337,-81.544,-36.222,179.837,5.198,148.947
C00695=1240.342,-81.794,-36.211,179.835,5.198,148.947
C00696=1240.347,-82.044,-36.199,179.833,5.198,148.948
C00697=1240.352,-82.294,-36.188,179.831,5.198,148.949
C00698=1240.358,-82.543,-36.177,179.828,5.198,148.950
C00699=1240.363,-82.793,-36.165,179.826,5.198,148.950
C00700=1240.368,-83.043,-36.153,179.823,5.198,148.951
C00701=1240.373,-83.292,-36.142,179.821,5.198,148.952
C00702=1240.378,-83.542,-36.130,179.818,5.198,148.952
C00703=1240.384,-83.791,-36.119,179.816,5.198,148.953
C00704=1240.389,-84.041,-36.108,179.814,5.198,148.954
C00705=1240.394,-84.291,-36.096,179.812,5.198,148.955
C00706=1240.399,-84.541,-36.084,179.809,5.197,148.955
C00707=1240.404,-84.790,-36.073,179.807,5.198,148.956
C00708=1240.409,-85.040,-36.062,179.804,5.197,148.957
C00709=1240.415,-85.289,-36.050,179.802,5.198,148.957
C00710=1240.420,-85.539,-36.040,179.799,5.198,148.958
C00711=1240.425,-85.789,-36.028,179.797,5.198,148.959
C00712=1240.430,-86.039,-36.016,179.794,5.197,148.960
C00713=1240.435,-86.288,-36.006,179.792,5.198,148.960
C00714=1240.440,-86.538,-35.994,179.789,5.197,148.961
C00715=1240.445,-86.787,-35.982,179.787,5.198,148.962
C00716=1240.451,-87.037,-35.970,179.785,5.198,148.963
C00717=1240.456,-87.288,-35.960,179.782,5.197,148.963
C00718=1240.461,-87.537,-35.949,179.780,5.198,148.964
C00719=1240.466,-87.787,-35.937,179.778,5.197,148.965
C00720=1240.471,-88.036,-35.926,179.776,5.198,148.965
C00721=1240.476,-88.286,-35.914,179.773,5.197,148.966
C00722=1240.482,-88.536,-35.904,179.771,5.198,148.967
C00723=1240.487,-88.785,-35.892,179.768,5.197,148.968
C00724=1240.492,-89.035,-35.881,179.766,5.197,148.968
C00725=1240.497,-89.285,-35.869,179.763,5.197,148.969
C00726=1240.502,-89.534,-35.858,179.761,5.197,148.970
C00727=1240.508,-89.784,-35.847,179.759,5.197,148.970
C00728=1240.513,-90.034,-35.836,179.757,5.197,148.971
C00729=1240.517,-90.284,-35.825,179.754,5.197,148.972
C00730=1240.523,-90.533,-35.813,179.752,5.197,148.973
C00731=1240.528,-90.783,-35.802,179.749,5.197,148.973
C00732=1240.533,-91.033,-35.791,179.747,5.197,148.974
C00733=1240.539,-91.282,-35.780,179.744,5.197,148.975
C00734=1240.544,-91.532,-35.769,179.742,5.197,148.976
C00735=1240.549,-91.782,-35.758,179.740,5.198,148.976
C00736=1240.553,-92.031,-35.747,179.737,5.197,148.977
C00737=1240.560,-92.281,-35.736,179.735,5.198,148.978
C00738=1240.564,-92.531,-35.724,179.732,5.197,148.978
C00739=1240.569,-92.780,-35.713,179.730,5.197,148.979
C00740=1240.575,-93.030,-35.702,179.727,5.197,148.980
C00741=1240.580,-93.280,-35.691,179.725,5.197,148.981
C00742=1240.585,-93.530,-35.680,179.723,5.197,148.981
C00743=1240.590,-93.779,-35.670,179.721,5.197,148.982
C00744=1240.596,-94.029,-35.658,179.718,5.197,148.983
C00745=1240.601,-94.279,-35.646,179.716,5.197,148.983
C00746=1240.606,-94.528,-35.636,179.713,5.197,148.984
C00747=1240.611,-94.778,-35.625,179.711,5.197,148.985
C00748=1240.616,-95.028,-35.613,179.708,5.196,148.986
C00749=1240.622,-95.277,-35.603,179.706,5.197,148.986
C00750=1240.627,-95.527,-35.592,179.704,5.197,148.987
C00751=1240.632,-95.777,-35.581,179.701,5.197,148.988
C00752=1240.638,-96.026,-35.569,179.699,5.197,148.988
C00753=1240.642,-96.276,-35.558,179.697,5.197,148.989
C00754=1240.647,-96.526,-35.548,179.695,5.197,148.990
C00755=1240.653,-96.775,-35.537,179.692,5.197,148.991
C00756=1240.658,-97.025,-35.526,179.690,5.197,148.991
C00757=1240.664,-97.275,-35.515,179.687,5.196,148.992
C00758=1240.669,-97.525,-35.504,179.685,5.197,148.993
C00759=1240.673,-97.775,-35.493,179.682,5.196,148.993
C00760=1240.679,-98.024,-35.482,179.680,5.197,148.994
C00761=1240.684,-98.274,-35.471,179.678,5.196,148.995
C00762=1240.689,-98.524,-35.461,179.676,5.197,148.996
C00763=1240.695,-98.773,-35.449,179.673,5.197,148.996
C00764=1240.699,-99.023,-35.438,179.671,5.196,148.997
C00765=1240.705,-99.272,-35.428,179.669,5.197,148.998
C00766=1240.710,-99.523,-35.417,179.666,5.196,148.998
C00767=1240.715,-99.772,-35.406,179.664,5.197,148.999
C00768=1240.721,-100.043,-35.394,179.661,5.197,149.000
C00769=1240.726,-100.313,-35.382,179.659,5.197,149.001
C00770=1240.732,-100.585,-35.371,179.656,5.197,149.002
C00771=1240.738,-100.855,-35.359,179.653,5.196,149.002
C00772=1240.743,-101.105,-35.348,179.651,5.196,149.003
C00773=1240.748,-101.355,-35.337,179.648,5.196,149.004
C00774=1240.753,-101.605,-35.327,179.646,5.196,149.004
C00775=1240.758,-101.854,-35.315,179.644,5.197,149.005
C00776=1240.763,-102.104,-35.305,179.642,5.196,149.006
C00777=1240.768,-102.353,-35.294,179.640,5.197,149.007
C00778=1240.774,-102.603,-35.284,179.637,5.196,149.007
C00779=1240.779,-102.853,-35.273,179.634,5.197,149.008
C00780=1240.784,-103.103,-35.261,179.632,5.196,149.009
C00781=1240.790,-103.353,-35.251,179.629,5.197,149.010
C00782=1240.794,-103.602,-35.240,179.627,5.196,149.010
C00783=1240.800,-103.852,-35.230,179.625,5.197,149.011
C00784=1240.805,-104.102,-35.219,179.622,5.196,149.012
C00785=1240.810,-104.351,-35.208,179.620,5.197,149.012
C00786=1240.815,-104.601,-35.197,179.618,5.197,149.013
C00787=1240.821,-104.851,-35.187,179.615,5.197,149.014
C00788=1240.826,-105.100,-35.176,179.613,5.197,149.015
C00789=1240.831,-105.350,-35.166,179.610,5.196,149.015
C00790=1240.836,-105.600,-35.155,179.608,5.197,149.016
C00791=1240.841,-105.849,-35.144,179.606,5.196,149.017
C00792=1240.846,-106.099,-35.134,179.604,5.197,149.017
C00793=1240.851,-106.350,-35.123,179.601,5.196,149.018
C00794=1240.857,-106.598,-35.112,179.599,5.197,149.019
C00795=1240.862,-106.849,-35.102,179.596,5.196,149.020
C00796=1240.867,-107.098,-35.091,179.594,5.196,149.020
C00797=1240.872,-107.348,-35.080,179.592,5.197,149.021
C00798=1240.878,-107.597,-35.070,179.589,5.196,149.022
C00799=1240.883,-107.848,-35.059,179.587,5.197,149.022
C00800=1240.888,-108.097,-35.049,179.584,5.196,149.023
C00801=1240.893,-108.347,-35.038,179.583,5.196,149.024
C00802=1240.899,-108.596,-35.028,179.580,5.196,149.024
C00803=1240.904,-108.847,-35.017,179.578,5.196,149.025
C00804=1240.909,-109.096,-35.007,179.575,5.196,149.026
C00805=1240.915,-109.346,-34.997,179.573,5.196,149.027
C00806=1240.919,-109.595,-34.985,179.571,5.196,149.027
C00807=1240.925,-109.845,-34.975,179.569,5.196,149.028
C00808=1240.930,-110.095,-34.965,179.566,5.196,149.029
C00809=1240.936,-110.345,-34.954,179.564,5.196,149.029
C00810=1240.940,-110.594,-34.943,179.562,5.196,149.030
C00811=1240.946,-110.844,-34.933,179.559,5.196,149.031
C00812=1240.950,-111.094,-34.923,179.557,5.196,149.032
C00813=1240.956,-111.343,-34.913,179.554,5.196,149.032
C00814=1240.961,-111.594,-34.902,179.552,5.196,149.033
C00815=1240.966,-111.843,-34.892,179.550,5.196,149.034
C00816=1240.972,-112.092,-34.881,179.547,5.196,149.034
C00817=1240.977,-112.342,-34.870,179.545,5.196,149.035
C00818=1240.982,-112.592,-34.860,179.543,5.196,149.036
C00819=1240.987,-112.842,-34.850,179.540,5.196,149.037
C00820=1240.993,-113.092,-34.839,179.538,5.196,149.037
C00821=1240.998,-113.342,-34.829,179.536,5.196,149.038
C00822=1241.003,-113.591,-34.819,179.533,5.196,149.039
C00823=1241.008,-113.841,-34.809,179.531,5.196,149.039
C00824=1241.013,-114.091,-34.798,179.529,5.197,149.040
C00825=1241.019,-114.340,-34.787,179.526,5.196,149.041
C00826=1241.024,-114.590,-34.777,179.524,5.196,149.042
C00827=1241.029,-114.840,-34.767,179.521,5.196,149.042
C00828=1241.035,-115.089,-34.756,179.519,5.196,149.043
C00829=1241.039,-115.339,-34.746,179.517,5.196,149.044
C00830=1241.045,-115.589,-34.736,179.515,5.196,149.044
C00831=1241.050,-115.839,-34.726,179.512,5.196,149.045
C00832=1241.055,-116.088,-34.715,179.510,5.196,149.046
C00833=1241.061,-116.338,-34.705,179.508,5.197,149.047
C00834=1241.066,-116.588,-34.695,179.505,5.196,149.047
C00835=1241.071,-116.837,-34.685,179.503,5.196,149.048
C00836=1241.076,-117.088,-34.675,179.500,5.196,149.049
C00837=1241.081,-117.337,-34.664,179.498,5.196,149.049
C00838=1241.087,-117.587,-34.654,179.495,5.196,149.050
C00839=1241.091,-117.837,-34.644,179.493,5.196,149.051
C00840=1241.097,-118.086,-34.634,179.491,5.196,149.052
C00841=1241.102,-118.336,-34.624,179.489,5.196,149.052
C00842=1241.107,-118.586,-34.613,179.487,5.196,149.053
C00843=1241.113,-118.836,-34.603,179.484,5.196,149.053
C00844=1241.118,-119.085,-34.593,179.482,5.196,149.054
C00845=1241.123,-119.335,-34.583,179.479,5.196,149.055
C00846=1241.128,-119.585,-34.573,179.477,5.196,149.056
C00847=1241.134,-119.834,-34.562,179.475,5.196,149.056
C00848=1241.138,-120.084,-34.552,179.473,5.196,149.057
C00849=1241.144,-120.334,-34.542,179.470,5.196,149.058
C00850=1241.149,-120.583,-34.532,179.468,5.196,149.059
C00851=1241.154,-120.833,-34.521,179.466,5.196,149.059
C00852=1241.160,-121.083,-34.512,179.463,5.196,149.060
C00853=1241.165,-121.333,-34.502,179.461,5.196,149.061
C00854=1241.170,-121.583,-34.492,179.458,5.196,149.061
C00855=1241.175,-121.832,-34.482,179.456,5.196,149.062
C00856=1241.181,-122.082,-34.472,179.453,5.196,149.063
C00857=1241.186,-122.332,-34.461,179.451,5.196,149.064
C00858=1241.191,-122.582,-34.451,179.449,5.196,149.064
C00859=1241.196,-122.831,-34.441,179.447,5.196,149.065
C00860=1241.201,-123.082,-34.432,179.445,5.196,149.066
C00861=1241.207,-123.331,-34.421,179.442,5.196,149.066
C00862=1241.212,-123.580,-34.412,179.440,5.196,149.067
C00863=1241.218,-123.830,-34.402,179.438,5.196,149.068
C00864=1241.222,-124.080,-34.391,179.435,5.196,149.068
C00865=1241.227,-124.329,-34.381,179.433,5.195,149.069
C00866=1241.233,-124.580,-34.372,179.431,5.196,149.070
C00867=1241.238,-124.830,-34.361,179.429,5.196,149.070
C00868=1241.243,-125.079,-34.352,179.426,5.196,149.071
C00869=1241.249,-125.329,-34.341,179.424,5.196,149.072
C00870=1241.254,-125.578,-34.332,179.421,5.196,149.073
C00871=1241.259,-125.829,-34.322,179.419,5.196,149.073
C00872=1240.837,-125.839,-34.356,179.415,5.200,149.075
C00873=1240.832,-125.589,-34.367,179.417,5.199,149.075
C00874=1240.827,-125.340,-34.376,179.419,5.200,149.074
C00875=1240.822,-125.090,-34.387,179.421,5.199,149.073
C00876=1240.817,-124.840,-34.396,179.424,5.199,149.073
C00877=1240.811,-124.590,-34.406,179.426,5.199,149.072
C00878=1240.805,-124.341,-34.416,179.428,5.199,149.071
C00879=1240.801,-124.091,-34.426,179.431,5.199,149.070
C00880=1240.796,-123.841,-34.436,179.433,5.199,149.070
C00881=1240.790,-123.592,-34.446,179.436,5.199,149.069
C00882=1240.785,-123.341,-34.456,179.438,5.199,149.068
C00883=1240.780,-123.091,-34.466,179.441,5.200,149.068
C00884=1240.774,-122.842,-34.476,179.443,5.199,149.067
C00885=1240.769,-122.593,-34.486,179.444,5.199,149.066
C00886=1240.764,-122.342,-34.496,179.447,5.200,149.066
C00887=1240.759,-122.093,-34.507,179.449,5.199,149.065
C00888=1240.753,-121.843,-34.517,179.452,5.200,149.064
C00889=1240.749,-121.593,-34.526,179.454,5.199,149.064
C00890=1240.743,-121.343,-34.536,179.456,5.200,149.063
C00891=1240.737,-121.094,-34.546,179.459,5.199,149.062
C00892=1240.733,-120.844,-34.556,179.461,5.199,149.061
C00893=1240.728,-120.594,-34.567,179.463,5.199,149.061
C00894=1240.722,-120.345,-34.577,179.465,5.199,149.060
C00895=1240.717,-120.094,-34.587,179.468,5.200,149.059
C00896=1240.712,-119.845,-34.597,179.470,5.199,149.058
C00897=1240.706,-119.596,-34.607,179.473,5.200,149.058
C00898=1240.701,-119.345,-34.618,179.475,5.199,149.057
C00899=1240.696,-119.096,-34.628,179.478,5.200,149.056
C00900=1240.691,-118.847,-34.638,179.480,5.199,149.056
C00901=1240.686,-118.596,-34.648,179.482,5.199,149.055
C00902=1240.680,-118.346,-34.658,179.485,5.199,149.054
C00903=1240.675,-118.097,-34.668,179.487,5.199,149.053
C00904=1240.670,-117.847,-34.678,179.489,5.199,149.053
C00905=1240.665,-117.597,-34.688,179.491,5.199,149.052
C00906=1240.659,-117.348,-34.698,179.494,5.200,149.052
C00907=1240.654,-117.097,-34.709,179.496,5.200,149.051
C00908=1240.648,-116.848,-34.719,179.498,5.200,149.050
C00909=1240.644,-116.598,-34.729,179.500,5.200,149.049
C00910=1240.639,-116.348,-34.739,179.503,5.199,149.049
C00911=1240.633,-116.100,-34.750,179.505,5.200,149.048
C00912=1240.628,-115.849,-34.761,179.507,5.199,149.047
C00913=1240.623,-115.600,-34.771,179.510,5.200,149.047
C00914=1240.618,-115.351,-34.781,179.512,5.199,149.046
C00915=1240.613,-115.100,-34.791,179.515,5.200,149.045
C00916=1240.607,-114.851,-34.801,179.517,5.199,149.044
C00917=1240.602,-114.600,-34.812,179.520,5.200,149.044
C00918=1240.597,-114.351,-34.822,179.522,5.200,149.043
C00919=1240.591,-114.101,-34.832,179.524,5.199,149.042
C00920=1240.586,-113.851,-34.843,179.526,5.200,149.042
C00921=1240.581,-113.602,-34.853,179.529,5.199,149.041
C00922=1240.576,-113.352,-34.863,179.531,5.200,149.040
C00923=1240.571,-113.102,-34.873,179.533,5.199,149.039
C00924=1240.566,-112.852,-34.884,179.536,5.200,149.039
C00925=1240.560,-112.603,-34.895,179.538,5.199,149.038
C00926=1240.555,-112.353,-34.905,179.541,5.200,149.037
C00927=1240.550,-112.103,-34.916,179.543,5.200,149.037
C00928=1240.544,-111.854,-34.926,179.545,5.199,149.036
C00929=1240.539,-111.603,-34.936,179.548,5.200,149.035
C00930=1240.534,-111.354,-34.946,179.550,5.199,149.034
C00931=1240.529,-111.104,-34.957,179.552,5.200,149.034
C00932=1240.524,-110.855,-34.967,179.554,5.199,149.033
C00933=1240.518,-110.605,-34.978,179.557,5.200,149.032
C00934=1240.513,-110.355,-34.988,179.559,5.199,149.032
C00935=1240.508,-110.106,-34.998,179.562,5.200,149.031
C00936=1240.503,-109.855,-35.009,179.564,5.200,149.030
C00937=1240.498,-109.606,-35.020,179.566,5.199,149.029
C00938=1240.493,-109.356,-35.031,179.569,5.200,149.029
C00939=1240.487,-109.107,-35.041,179.571,5.199,149.028
C00940=1240.482,-108.856,-35.051,179.574,5.200,149.027
C00941=1240.476,-108.607,-35.062,179.576,5.199,149.026
C00942=1240.472,-108.357,-35.073,179.578,5.200,149.026
C00943=1240.466,-108.108,-35.083,179.580,5.199,149.025
C00944=1240.461,-107.857,-35.094,179.583,5.200,149.025
C00945=1240.455,-107.608,-35.104,179.585,5.200,149.024
C00946=1240.451,-107.358,-35.115,179.587,5.200,149.023
C00947=1240.445,-107.109,-35.125,179.590,5.200,149.022
C00948=1240.440,-106.859,-35.136,179.592,5.200,149.022
C00949=1240.435,-106.610,-35.147,179.594,5.200,149.021
C00950=1240.430,-106.359,-35.157,179.596,5.200,149.020
C00951=1240.424,-106.110,-35.168,179.599,5.200,149.020
C00952=1240.419,-105.860,-35.178,179.601,5.200,149.019
C00953=1240.414,-105.611,-35.189,179.604,5.200,149.018
C00954=1240.409,-105.360,-35.200,179.606,5.200,149.017
C00955=1240.403,-105.111,-35.210,179.609,5.200,149.017
C00956=1240.399,-104.861,-35.221,179.611,5.200,149.016
C00957=1240.393,-104.612,-35.231,179.613,5.200,149.015
C00958=1240.388,-104.361,-35.242,179.615,5.200,149.015
C00959=1240.383,-104.113,-35.253,179.618,5.200,149.014
C00960=1240.378,-103.862,-35.263,179.620,5.200,149.013
C00961=1240.373,-103.613,-35.275,179.622,5.200,149.012
C00962=1240.367,-103.363,-35.285,179.625,5.200,149.012
C00963=1240.362,-103.113,-35.296,179.627,5.200,149.011
C00964=1240.357,-102.864,-35.306,179.630,5.200,149.010
C00965=1240.352,-102.614,-35.317,179.632,5.200,149.010
C00966=1240.347,-102.364,-35.327,179.635,5.200,149.009
C00967=1240.342,-102.115,-35.339,179.637,5.200,149.008
C00968=1240.336,-101.865,-35.349,179.639,5.201,149.007
C00969=1240.332,-101.615,-35.360,179.641,5.200,149.007
C00970=1240.326,-101.365,-35.371,179.644,5.200,149.006
C00971=1240.321,-101.116,-35.382,179.646,5.200,149.005
C00972=1240.316,-100.866,-35.393,179.649,5.200,149.004
C00973=1240.310,-100.596,-35.404,179.651,5.200,149.004
C00974=1240.305,-100.325,-35.416,179.654,5.200,149.003
C00975=1240.299,-100.053,-35.428,179.656,5.200,149.002
C00976=1240.293,-99.783,-35.439,179.659,5.200,149.001
C00977=1240.288,-99.533,-35.450,179.662,5.200,149.001
C00978=1240.283,-99.283,-35.462,179.664,5.200,149.000
C00979=1240.277,-99.033,-35.472,179.666,5.200,148.999
C00980=1240.272,-98.784,-35.483,179.669,5.200,148.998
C00981=1240.267,-98.533,-35.494,179.671,5.200,148.998
C00982=1240.262,-98.285,-35.505,179.673,5.200,148.997
C00983=1240.257,-98.035,-35.516,179.676,5.200,148.996
C00984=1240.251,-97.785,-35.527,179.678,5.200,148.996
C00985=1240.246,-97.535,-35.538,179.681,5.200,148.995
C00986=1240.241,-97.285,-35.548,179.683,5.200,148.994
C00987=1240.236,-97.036,-35.559,179.685,5.200,148.993
C00988=1240.231,-96.786,-35.570,179.687,5.200,148.993
C00989=1240.225,-96.537,-35.582,179.690,5.200,148.992
C00990=1240.220,-96.287,-35.592,179.692,5.200,148.991
C00991=1240.215,-96.037,-35.603,179.695,5.201,148.991
C00992=1240.210,-95.787,-35.614,179.697,5.200,148.990
C00993=1240.205,-95.538,-35.625,179.700,5.201,148.989
C00994=1240.200,-95.288,-35.637,179.702,5.200,148.988
C00995=1240.194,-95.038,-35.647,179.704,5.200,148.988
C00996=1240.189,-94.789,-35.658,179.707,5.200,148.987
C00997=1240.184,-94.538,-35.669,179.709,5.200,148.986
C00998=1240.178,-94.289,-35.680,179.711,5.201,148.986
C00999=1240.174,-94.040,-35.692,179.713,5.200,148.985
C01000=1240.169,-93.789,-35.702,179.716,5.201,148.984
C01001=1240.163,-93.540,-35.713,179.718,5.200,148.983
C01002=1240.158,-93.290,-35.725,179.721,5.201,148.983
C01003=1240.153,-93.040,-35.736,179.723,5.200,148.982
C01004=1240.148,-92.791,-35.747,179.726,5.201,148.981
C01005=1240.143,-92.542,-35.758,179.728,5.201,148.981
C01006=1240.137,-92.291,-35.769,179.730,5.201,148.980
C01007=1240.133,-92.041,-35.780,179.732,5.201,148.979
C01008=1240.127,-91.793,-35.791,179.735,5.201,148.978
C01009=1240.121,-91.542,-35.802,179.737,5.201,148.978
C01010=1240.117,-91.292,-35.814,179.739,5.200,148.977
C01011=1240.112,-91.043,-35.825,179.742,5.201,148.976
C01012=1240.107,-90.793,-35.835,179.744,5.200,148.976
C01013=1240.101,-90.543,-35.847,179.747,5.201,148.975
C01014=1240.096,-90.294,-35.858,179.749,5.201,148.974
C01015=1240.091,-90.045,-35.869,179.752,5.201,148.973
C01016=1240.085,-89.794,-35.880,179.754,5.200,148.973
C01017=1240.081,-89.545,-35.892,179.757,5.201,148.972
C01018=1240.075,-89.296,-35.903,179.759,5.200,148.971
C01019=1240.070,-89.046,-35.915,179.762,5.201,148.970
C01020=1240.065,-88.795,-35.925,179.764,5.201,148.970
C01021=1240.060,-88.546,-35.936,179.766,5.201,148.969
C01022=1240.054,-88.297,-35.948,179.768,5.201,148.968
C01023=1240.050,-88.047,-35.959,179.771,5.201,148.968
C01024=1240.044,-87.797,-35.971,179.773,5.201,148.967
C01025=1240.039,-87.547,-35.982,179.776,5.201,148.966
C01026=1240.034,-87.298,-35.993,179.778,5.201,148.965
C01027=1240.028,-87.048,-36.004,179.780,5.201,148.965
C01028=1240.024,-86.798,-36.016,179.783,5.201,148.964
C01029=1240.019,-86.549,-36.027,179.785,5.201,148.963
C01030=1240.013,-86.299,-36.039,179.787,5.201,148.963
C01031=1240.008,-86.049,-36.049,179.790,5.201,148.962
C01032=1240.003,-85.799,-36.061,179.792,5.201,148.961
C01033=1239.998,-85.550,-36.072,179.794,5.201,148.960
C01034=1239.993,-85.300,-36.084,179.797,5.201,148.960
C01035=1239.987,-85.051,-36.095,179.799,5.201,148.959
C01036=1239.982,-84.801,-36.106,179.802,5.202,148.958
C01037=1239.977,-84.551,-36.118,179.804,5.201,148.958
C01038=1239.972,-84.302,-36.130,179.807,5.202,148.957
C01039=1239.967,-84.051,-36.141,179.809,5.201,148.956
C01040=1239.961,-83.802,-36.152,179.812,5.201,148.955
C01041=1239.957,-83.552,-36.163,179.814,5.201,148.955
C01042=1239.951,-83.303,-36.175,179.817,5.202,148.954
C01043=1239.946,-83.053,-36.186,179.819,5.201,148.953
C01044=1239.941,-82.803,-36.198,179.821,5.202,148.952
C01045=1239.936,-82.553,-36.209,179.823,5.201,148.952
C01046=1239.930,-82.304,-36.221,179.826,5.202,148.951
C01047=1239.926,-82.054,-36.232,179.828,5.201,148.950
C01048=1239.920,-81.805,-36.244,179.831,5.202,148.950
C01049=1239.916,-81.555,-36.255,179.833,5.202,148.949
C01050=1239.910,-81.305,-36.267,179.836,5.202,148.948
C01051=1239.905,-81.055,-36.278,179.838,5.202,148.947
C01052=1239.899,-80.806,-36.290,179.840,5.201,148.947
C01053=1239.895,-80.557,-36.301,179.842,5.202,148.946
C01054=1239.889,-80.307,-36.313,179.845,5.201,148.945
C01055=1239.885,-80.057,-36.324,179.847,5.202,148.945
C01056=1239.879,-79.807,-36.336,179.849,5.202,148.944
C01057=1239.874,-79.557,-36.348,179.852,5.202,148.943
C01058=1239.869,-79.307,-36.360,179.855,5.201,148.942
C01059=1239.864,-79.059,-36.370,179.857,5.202,148.942
C01060=1239.858,-78.809,-36.382,179.859,5.202,148.941
C01061=1239.853,-78.559,-36.394,179.862,5.202,148.940
C01062=1239.848,-78.309,-36.406,179.864,5.202,148.939
C01063=1239.843,-78.059,-36.417,179.867,5.202,148.939
C01064=1239.838,-77.809,-36.429,179.869,5.202,148.938
C01065=1239.833,-77.560,-36.441,179.872,5.202,148.937
C01066=1239.828,-77.310,-36.452,179.874,5.202,148.937
C01067=1239.822,-77.061,-36.464,179.876,5.202,148.936
C01068=1239.817,-76.811,-36.476,179.878,5.202,148.935
C01069=1239.812,-76.562,-36.487,179.881,5.203,148.934
C01070=1239.807,-76.312,-36.499,179.883,5.202,148.934
C01071=1239.802,-76.062,-36.510,179.886,5.203,148.933
C01072=1239.797,-75.812,-36.522,179.888,5.202,148.932
C01073=1239.791,-75.562,-36.534,179.891,5.203,148.932
C01074=1239.786,-75.313,-36.546,179.893,5.202,148.931
C01075=1239.781,-75.063,-36.558,179.896,5.203,148.930
C01076=1239.776,-74.813,-36.570,179.898,5.202,148.929
C01077=1239.770,-74.544,-36.583,179.901,5.203,148.929
C01078=1239.764,-74.273,-36.595,179.903,5.202,148.928
C01079=1239.759,-74.002,-36.608,179.906,5.202,148.927
C01080=1239.753,-73.733,-36.620,179.909,5.203,148.926
C01081=1239.748,-73.483,-36.632,179.911,5.203,148.925
C01082=1239.743,-73.234,-36.644,179.913,5.203,148.925
C01083=1239.738,-72.984,-36.656,179.915,5.203,148.924
C01084=1239.733,-72.734,-36.667,179.918,5.203,148.923
C01085=1239.728,-72.484,-36.679,179.920,5.203,148.923
C01086=1239.722,-72.234,-36.691,179.923,5.203,148.922
C01087=1239.718,-71.985,-36.703,179.925,5.203,148.921
C01088=1239.712,-71.735,-36.715,179.928,5.204,148.921
C01089=1239.707,-71.485,-36.727,179.930,5.203,148.920
C01090=1239.702,-71.236,-36.738,179.933,5.203,148.919
C01091=1239.697,-70.987,-36.751,179.935,5.203,148.918
C01092=1239.692,-70.737,-36.763,179.938,5.203,148.917
C01093=1239.686,-70.487,-36.775,179.940,5.203,148.917
C01094=1239.682,-70.238,-36.787,179.942,5.204,148.916
C01095=1239.677,-69.988,-36.799,179.944,5.203,148.915
C01096=1239.671,-69.738,-36.810,179.947,5.204,148.915
C01097=1239.666,-69.488,-36.822,179.949,5.203,148.914
C01098=1239.661,-69.239,-36.834,179.952,5.204,148.913
C01099=1239.656,-68.989,-36.846,179.954,5.204,148.912
C01100=1239.650,-68.739,-36.858,179.957,5.204,148.912
C01101=1239.645,-68.490,-36.871,179.959,5.204,148.911
C01102=1239.641,-68.240,-36.882,179.961,5.204,148.910
C01103=1239.635,-67.990,-36.894,179.964,5.204,148.910
C01104=1239.630,-67.741,-36.907,179.966,5.204,148.909
C01105=1239.625,-67.491,-36.918,179.969,5.204,148.908
C01106=1239.620,-67.242,-36.930,179.971,5.204,148.907
C01107=1239.615,-66.992,-36.942,179.974,5.204,148.907
C01108=1239.609,-66.742,-36.954,179.976,5.204,148.906
C01109=1239.604,-66.493,-36.967,179.978,5.204,148.905
C01110=1239.599,-66.243,-36.979,179.981,5.204,148.904
C01111=1239.594,-65.994,-36.991,179.983,5.204,148.904
C01112=1239.589,-65.744,-37.003,179.986,5.205,148.903
C01113=1239.584,-65.494,-37.014,179.988,5.204,148.902
C01114=1239.578,-65.245,-37.027,179.990,5.205,148.902
C01115=1239.573,-64.995,-37.039,179.993,5.204,148.901
C01116=1239.568,-64.745,-37.052,179.995,5.205,148.900
C01117=1239.563,-64.496,-37.063,179.997,5.205,148.900
C01118=1239.558,-64.246,-37.075,-179.999,5.205,148.899
C01119=1239.553,-63.996,-37.087,-179.997,5.204,148.898
C01120=1239.548,-63.747,-37.100,-179.995,5.205,148.897
C01121=1239.543,-63.496,-37.112,-179.993,5.204,148.896
C01122=1239.537,-63.246,-37.124,-179.990,5.205,148.896
C01123=1239.533,-62.997,-37.136,-179.988,5.205,148.895
C01124=1239.527,-62.748,-37.148,-179.985,5.205,148.894
C01125=1239.522,-62.498,-37.161,-179.983,5.205,148.894
C01126=1239.517,-62.249,-37.173,-179.980,5.205,148.893
C01127=1239.512,-61.999,-37.185,-179.978,5.206,148.892
C01128=1239.507,-61.750,-37.198,-179.976,5.205,148.892
C01129=1239.501,-61.500,-37.209,-179.973,5.206,148.891
C01130=1239.496,-61.250,-37.222,-179.971,5.206,148.890
C01131=1239.491,-61.000,-37.234,-179.968,5.206,148.889
C01132=1239.487,-60.751,-37.246,-179.966,5.205,148.888
C01133=1239.481,-60.501,-37.258,-179.963,5.206,148.888
C01134=1239.476,-60.252,-37.271,-179.961,5.206,148.887
C01135=1239.471,-60.002,-37.283,-179.958,5.206,148.886
C01136=1239.466,-59.752,-37.295,-179.956,5.206,148.886
C01137=1239.461,-59.503,-37.308,-179.954,5.206,148.885
C01138=1239.455,-59.253,-37.320,-179.951,5.206,148.884
C01139=1239.451,-59.003,-37.333,-179.949,5.206,148.884
C01140=1239.445,-58.753,-37.345,-179.947,5.206,148.883
C01141=1239.440,-58.504,-37.357,-179.944,5.206,148.882
C01142=1239.435,-58.254,-37.370,-179.942,5.206,148.881
C01143=1239.430,-58.004,-37.382,-179.939,5.206,148.881
C01144=1239.425,-57.755,-37.394,-179.937,5.206,148.880
C01145=1239.419,-57.506,-37.407,-179.934,5.206,148.879
C01146=1239.415,-57.255,-37.419,-179.932,5.206,148.878
C01147=1239.409,-57.006,-37.432,-179.929,5.207,148.878
C01148=1239.404,-56.757,-37.444,-179.927,5.207,148.877
C01149=1239.399,-56.507,-37.456,-179.924,5.207,148.876
C01150=1239.394,-56.257,-37.469,-179.922,5.207,148.876
C01151=1239.389,-56.007,-37.482,-179.920,5.207,148.875
C01152=1239.384,-55.757,-37.494,-179.917,5.207,148.874
C01153=1239.379,-55.508,-37.506,-179.915,5.207,148.873
C01154=1239.374,-55.259,-37.519,-179.912,5.208,148.873
C01155=1239.368,-55.009,-37.532,-179.910,5.207,148.872
C01156=1239.363,-54.759,-37.543,-179.907,5.207,148.871
C01157=1239.358,-54.509,-37.556,-179.905,5.207,148.870
C01158=1239.353,-54.260,-37.569,-179.902,5.208,148.870
C01159=1239.348,-54.010,-37.581,-179.900,5.207,148.869
C01160=1239.343,-53.761,-37.593,-179.898,5.208,148.868
C01161=1239.338,-53.511,-37.606,-179.895,5.207,148.868
C01162=1239.333,-53.262,-37.619,-179.893,5.208,148.867
C01163=1239.328,-53.012,-37.632,-179.891,5.208,148.866
C01164=1239.323,-52.762,-37.644,-179.888,5.208,148.865
C01165=1239.317,-52.513,-37.656,-179.885,5.209,148.865
C01166=1239.313,-52.263,-37.669,-179.883,5.208,148.864
C01167=1239.308,-52.014,-37.682,-179.880,5.208,148.863
C01168=1239.302,-51.764,-37.695,-179.878,5.208,148.862
C01169=1239.297,-51.514,-37.707,-179.875,5.209,148.862
C01170=1239.292,-51.264,-37.720,-179.873,5.208,148.861
C01171=1239.287,-51.015,-37.732,-179.871,5.209,148.860
C01172=1239.282,-50.765,-37.745,-179.869,5.208,148.860
C01173=1239.277,-50.516,-37.758,-179.866,5.209,148.859
C01174=1239.272,-50.266,-37.771,-179.864,5.209,148.858
C01175=1239.267,-50.016,-37.782,-179.861,5.209,148.858
C01176=1239.262,-49.767,-37.795,-179.858,5.210,148.857
C01177=1239.256,-49.517,-37.808,-179.856,5.209,148.856
C01178=1239.251,-49.267,-37.821,-179.853,5.209,148.855
C01179=1239.246,-49.018,-37.834,-179.851,5.209,148.854
C01180=1239.241,-48.769,-37.846,-179.848,5.210,148.854
C01181=1239.236,-48.499,-37.860,-179.846,5.209,148.853
C01182=1239.230,-48.229,-37.874,-179.844,5.210,148.852
C01183=1239.225,-47.960,-37.888,-179.841,5.210,148.851
C01184=1239.219,-47.690,-37.902,-179.838,5.210,148.851
C01185=1239.214,-47.440,-37.915,-179.836,5.210,148.850
C01186=1239.209,-47.190,-37.927,-179.834,5.210,148.849
C01187=1239.204,-46.941,-37.940,-179.831,5.210,148.849
C01188=1239.198,-46.691,-37.953,-179.828,5.211,148.848
C01189=1239.193,-46.441,-37.965,-179.826,5.210,148.847
C01190=1239.188,-46.191,-37.978,-179.823,5.211,148.846
C01191=1239.183,-45.942,-37.991,-179.821,5.210,148.846
C01192=1239.178,-45.693,-38.003,-179.818,5.211,148.845
C01193=1239.173,-45.443,-38.017,-179.816,5.210,148.844
C01194=1239.168,-45.193,-38.029,-179.814,5.211,148.843
C01195=1239.163,-44.944,-38.042,-179.812,5.211,148.843
C01196=1239.158,-44.694,-38.055,-179.809,5.211,148.842
C01197=1239.152,-44.444,-38.068,-179.806,5.212,148.841
C01198=1239.147,-44.195,-38.081,-179.804,5.211,148.841
C01199=1239.143,-43.946,-38.095,-179.801,5.212,148.840
C01200=1239.138,-43.696,-38.107,-179.799,5.211,148.839
C01201=1239.132,-43.447,-38.120,-179.796,5.212,148.838
C01202=1239.127,-43.197,-38.133,-179.794,5.211,148.838
C01203=1239.122,-42.947,-38.146,-179.791,5.212,148.837
C01204=1239.118,-42.697,-38.159,-179.789,5.211,148.836
C01205=1239.112,-42.448,-38.172,-179.787,5.212,148.836
C01206=1239.107,-42.198,-38.185,-179.784,5.212,148.835
C01207=1239.102,-41.948,-38.198,-179.782,5.212,148.834
C01208=1239.096,-41.699,-38.211,-179.779,5.213,148.833
C01209=1239.091,-41.449,-38.223,-179.777,5.212,148.833
C01210=1239.087,-41.199,-38.236,-179.775,5.213,148.832
C01211=1239.081,-40.950,-38.250,-179.772,5.213,148.831
C01212=1239.077,-40.700,-38.263,-179.769,5.213,148.830
C01213=1239.071,-40.451,-38.276,-179.767,5.212,148.830
C01214=1239.066,-40.201,-38.289,-179.765,5.213,148.829
C01215=1239.061,-39.951,-38.302,-179.762,5.213,148.828
C01216=1239.056,-39.702,-38.315,-179.760,5.213,148.828
C01217=1239.051,-39.452,-38.328,-179.757,5.214,148.827
C01218=1239.046,-39.203,-38.342,-179.755,5.213,148.826
C01219=1239.041,-38.954,-38.354,-179.752,5.214,148.825
C01220=1239.035,-38.703,-38.368,-179.750,5.213,148.825
C01221=1239.030,-38.454,-38.380,-179.748,5.214,148.824
C01222=1239.026,-38.204,-38.393,-179.745,5.214,148.823
C01223=1239.020,-37.955,-38.407,-179.743,5.214,148.823
C01224=1239.015,-37.706,-38.420,-179.740,5.214,148.822
C01225=1239.010,-37.455,-38.433,-179.738,5.214,148.821
C01226=1239.005,-37.206,-38.446,-179.735,5.214,148.820
C01227=1239.001,-36.957,-38.460,-179.733,5.214,148.820
C01228=1238.995,-36.707,-38.473,-179.730,5.215,148.819
C01229=1238.990,-36.457,-38.486,-179.728,5.215,148.818
C01230=1238.984,-36.207,-38.499,-179.725,5.215,148.818
C01231=1238.979,-35.959,-38.512,-179.723,5.215,148.817
C01232=1238.974,-35.708,-38.526,-179.721,5.215,148.816
C01233=1238.969,-35.459,-38.538,-179.718,5.216,148.815
C01234=1238.965,-35.209,-38.551,-179.716,5.215,148.815
C01235=1238.959,-34.960,-38.565,-179.713,5.215,148.814
C01236=1238.954,-34.710,-38.578,-179.710,5.216,148.813
C01237=1238.949,-34.460,-38.591,-179.708,5.216,148.812
C01238=1238.944,-34.211,-38.605,-179.705,5.216,148.812
C01239=1238.939,-33.961,-38.618,-179.703,5.216,148.811
C01240=1238.934,-33.711,-38.631,-179.701,5.216,148.810
C01241=1238.928,-33.462,-38.645,-179.698,5.217,148.810
C01242=1238.924,-33.212,-38.658,-179.696,5.217,148.809
C01243=1238.918,-32.963,-38.671,-179.693,5.217,148.808
C01244=1238.914,-32.713,-38.685,-179.691,5.217,148.808
C01245=1238.908,-32.464,-38.698,-179.688,5.217,148.807
C01246=1238.903,-32.214,-38.711,-179.686,5.217,148.806
C01247=1238.898,-31.965,-38.725,-179.683,5.217,148.805
C01248=1238.893,-31.715,-38.738,-179.681,5.218,148.804
C01249=1238.888,-31.466,-38.752,-179.678,5.217,148.804
C01250=1238.883,-31.215,-38.765,-179.676,5.218,148.803
C01251=1238.878,-30.966,-38.779,-179.674,5.218,148.802
C01252=1238.873,-30.716,-38.792,-179.671,5.218,148.802
C01253=1238.867,-30.467,-38.805,-179.668,5.219,148.801
C01254=1238.863,-30.217,-38.819,-179.666,5.218,148.800
C01255=1238.857,-29.968,-38.832,-179.664,5.219,148.800
C01256=1238.853,-29.718,-38.846,-179.662,5.218,148.799
C01257=1238.847,-29.469,-38.859,-179.659,5.219,148.798
C01258=1238.842,-29.219,-38.873,-179.656,5.219,148.797
C01259=1238.838,-28.969,-38.886,-179.654,5.219,148.797
C01260=1238.832,-28.720,-38.900,-179.651,5.219,148.796
C01261=1238.828,-28.470,-38.913,-179.649,5.219,148.795
C01262=1238.822,-28.221,-38.927,-179.646,5.220,148.794
C01263=1238.818,-27.971,-38.940,-179.644,5.219,148.794
C01264=1238.812,-27.722,-38.954,-179.642,5.220,148.793
C01265=1238.807,-27.472,-38.967,-179.639,5.220,148.792
C01266=1238.802,-27.223,-38.981,-179.637,5.220,148.792
C01267=1238.797,-26.973,-38.994,-179.634,5.220,148.791
C01268=1238.792,-26.723,-39.008,-179.632,5.220,148.790
C01269=1238.787,-26.474,-39.021,-179.629,5.220,148.789
C01270=1238.782,-26.224,-39.035,-179.626,5.221,148.789
C01271=1238.777,-25.975,-39.048,-179.624,5.221,148.788
C01272=1238.772,-25.725,-39.062,-179.621,5.221,148.787
C01273=1238.767,-25.475,-39.076,-179.619,5.221,148.787
C01274=1238.761,-25.226,-39.089,-179.617,5.221,148.786
C01275=1238.757,-24.976,-39.103,-179.614,5.222,148.785
C01276=1238.751,-24.726,-39.117,-179.612,5.221,148.784
C01277=1238.746,-24.477,-39.130,-179.609,5.222,148.784
C01278=1238.742,-24.227,-39.145,-179.607,5.222,148.783
C01279=1238.736,-23.978,-39.158,-179.605,5.222,148.782
C01280=1238.731,-23.728,-39.171,-179.602,5.223,148.782
C01281=1238.726,-23.479,-39.185,-179.599,5.222,148.781
C01282=1238.721,-23.229,-39.199,-179.597,5.223,148.780
C01283=1238.716,-22.980,-39.213,-179.594,5.223,148.779
C01284=1238.711,-22.730,-39.226,-179.592,5.223,148.779
C01285=1238.705,-22.461,-39.241,-179.589,5.223,148.778
C01286=1238.700,-22.191,-39.256,-179.587,5.224,148.777
C01287=1238.694,-21.922,-39.271,-179.584,5.223,148.776
C01288=1238.690,-21.653,-39.285,-179.581,5.224,148.776
C01289=1238.684,-21.404,-39.299,-179.579,5.224,148.775
C01290=1238.679,-21.154,-39.313,-179.577,5.224,148.774
C01291=1238.673,-20.905,-39.327,-179.574,5.224,148.774
C01292=1238.669,-20.655,-39.340,-179.571,5.225,148.773
C01293=1238.664,-20.405,-39.354,-179.569,5.224,148.772
C01294=1238.658,-20.156,-39.368,-179.566,5.225,148.771
C01295=1238.653,-19.906,-39.383,-179.564,5.225,148.771
C01296=1238.649,-19.656,-39.396,-179.561,5.225,148.770
C01297=1238.643,-19.407,-39.410,-179.559,5.226,148.769
C01298=1238.638,-19.158,-39.424,-179.557,5.225,148.768
C01299=1238.633,-18.908,-39.438,-179.554,5.226,148.768
C01300=1238.628,-18.658,-39.452,-179.552,5.225,148.767
C01301=1238.623,-18.409,-39.465,-179.549,5.226,148.766
C01302=1238.618,-18.159,-39.479,-179.547,5.227,148.766
C01303=1238.614,-17.910,-39.494,-179.544,5.226,148.765
C01304=1238.608,-17.661,-39.507,-179.542,5.227,148.764
C01305=1238.603,-17.410,-39.521,-179.539,5.227,148.764
C01306=1238.598,-17.161,-39.535,-179.537,5.227,148.763
C01307=1238.593,-16.912,-39.549,-179.534,5.227,148.762
C01308=1238.588,-16.662,-39.563,-179.532,5.227,148.761
C01309=1238.583,-16.412,-39.577,-179.529,5.227,148.761
C01310=1238.578,-16.163,-39.591,-179.527,5.228,148.760
C01311=1238.572,-15.913,-39.605,-179.524,5.228,148.759
C01312=1238.567,-15.663,-39.619,-179.522,5.228,148.759
C01313=1238.563,-15.414,-39.633,-179.519,5.229,148.758
C01314=1238.558,-15.164,-39.647,-179.517,5.228,148.757
C01315=1238.553,-14.915,-39.661,-179.514,5.229,148.756
C01316=1238.548,-14.666,-39.675,-179.512,5.229,148.756
C01317=1238.543,-14.416,-39.689,-179.510,5.229,148.755
C01318=1238.538,-14.166,-39.704,-179.507,5.230,148.754
C01319=1238.532,-13.917,-39.717,-179.504,5.229,148.753
C01320=1238.527,-13.667,-39.732,-179.502,5.230,148.753
C01321=1238.523,-13.417,-39.745,-179.499,5.230,148.752
C01322=1238.518,-13.168,-39.759,-179.497,5.230,148.751
C01323=1238.512,-12.919,-39.773,-179.494,5.230,148.751
C01324=1238.507,-12.669,-39.787,-179.492,5.231,148.750
C01325=1238.502,-12.419,-39.801,-179.490,5.231,148.749
C01326=1238.497,-12.169,-39.816,-179.487,5.231,148.749
C01327=1238.492,-11.920,-39.830,-179.484,5.232,148.748
C01328=1238.487,-11.671,-39.844,-179.482,5.231,148.747
C01329=1238.482,-11.421,-39.858,-179.480,5.232,148.747
C01330=1238.477,-11.171,-39.873,-179.478,5.232,148.746
C01331=1238.472,-10.922,-39.887,-179.475,5.232,148.745
C01332=1238.466,-10.673,-39.901,-179.472,5.232,148.744
C01333=1238.461,-10.423,-39.915,-179.470,5.232,148.744
C01334=1238.456,-10.173,-39.929,-179.467,5.232,148.743
C01335=1238.451,-9.923,-39.944,-179.464,5.233,148.742
C01336=1238.446,-9.674,-39.958,-179.462,5.233,148.741
C01337=1238.442,-9.425,-39.973,-179.460,5.233,148.741
C01338=1238.437,-9.176,-39.986,-179.457,5.234,148.740
C01339=1238.432,-8.926,-40.000,-179.455,5.233,148.739
C01340=1238.427,-8.677,-40.015,-179.452,5.234,148.739
C01341=1238.422,-8.427,-40.029,-179.450,5.235,148.738
C01342=1238.417,-8.177,-40.043,-179.447,5.234,148.737
C01343=1238.412,-7.927,-40.058,-179.445,5.235,148.737
C01344=1238.406,-7.678,-40.072,-179.442,5.235,148.736
C01345=1238.401,-7.428,-40.086,-179.440,5.235,148.735
C01346=1238.396,-7.179,-40.101,-179.437,5.236,148.735
C01347=1238.391,-6.930,-40.116,-179.434,5.236,148.734
C01348=1238.386,-6.680,-40.130,-179.432,5.235,148.733
C01349=1238.381,-6.430,-40.144,-179.430,5.236,148.732
C01350=1238.377,-6.180,-40.158,-179.427,5.236,148.732
C01351=1238.371,-5.931,-40.172,-179.425,5.236,148.731
C01352=1238.366,-5.682,-40.187,-179.422,5.237,148.730
C01353=1238.361,-5.433,-40.202,-179.420,5.236,148.729
C01354=1238.356,-5.183,-40.216,-179.417,5.237,148.729
C01355=1238.351,-4.933,-40.230,-179.415,5.238,148.728
C01356=1238.347,-4.684,-40.244,-179.413,5.237,148.727
C01357=1238.342,-4.434,-40.259,-179.410,5.238,148.727
C01358=1238.337,-4.185,-40.274,-179.407,5.238,148.726
C01359=1238.332,-3.935,-40.288,-179.405,5.238,148.725
C01360=1238.326,-3.686,-40.302,-179.403,5.239,148.725
C01361=1238.321,-3.436,-40.317,-179.400,5.239,148.724
C01362=1238.316,-3.187,-40.332,-179.397,5.238,148.723
C01363=1238.311,-2.937,-40.346,-179.395,5.239,148.722
C01364=1238.306,-2.687,-40.360,-179.392,5.240,148.722
C01365=1238.301,-2.438,-40.375,-179.390,5.239,148.721
C01366=1238.297,-2.189,-40.390,-179.387,5.240,148.720
C01367=1238.292,-1.939,-40.404,-179.385,5.240,148.720
C01368=1238.286,-1.689,-40.419,-179.383,5.240,148.719
C01369=1238.281,-1.439,-40.433,-179.380,5.241,148.718
C01370=1238.276,-1.190,-40.448,-179.377,5.241,148.717
C01371=1238.271,-0.940,-40.462,-179.375,5.242,148.717
C01372=1238.266,-0.691,-40.477,-179.373,5.241,148.716
C01373=1238.261,-0.442,-40.491,-179.370,5.242,148.715
C01374=1238.255,-0.192,-40.506,-179.367,5.242,148.715
C01375=1238.250,0.057,-40.520,-179.365,5.242,148.714
C01376=1238.246,0.306,-40.535,-179.363,5.243,148.713
C01377=1238.241,0.556,-40.550,-179.360,5.243,148.713
C01378=1238.236,0.805,-40.565,-179.358,5.243,148.712
C01379=1238.231,1.055,-40.579,-179.355,5.243,148.711
C01380=1238.226,1.305,-40.594,-179.352,5.244,148.710
C01381=1238.221,1.554,-40.609,-179.350,5.243,148.710
C01382=1238.216,1.804,-40.623,-179.347,5.244,148.709
C01383=1238.210,2.054,-40.638,-179.345,5.244,148.708
C01384=1238.206,2.303,-40.653,-179.343,5.244,148.708
C01385=1238.201,2.553,-40.667,-179.340,5.245,148.707
C01386=1238.196,2.802,-40.682,-179.337,5.245,148.706
C01387=1238.190,3.052,-40.697,-179.335,5.245,148.706
C01388=1238.186,3.301,-40.712,-179.333,5.246,148.705
C01389=1238.181,3.570,-40.728,-179.330,5.246,148.704
C01390=1238.175,3.839,-40.744,-179.327,5.246,148.703
C01391=1238.170,4.108,-40.760,-179.324,5.247,148.703
C01392=1238.164,4.376,-40.775,-179.322,5.246,148.702
C01393=1238.159,4.626,-40.790,-179.319,5.247,148.701
C01394=1238.154,4.875,-40.805,-179.317,5.248,148.700
C01395=1238.149,5.125,-40.820,-179.315,5.247,148.700
C01396=1238.144,5.374,-40.835,-179.312,5.248,148.699
C01397=1238.139,5.624,-40.849,-179.309,5.248,148.698
C01398=1238.134,5.873,-40.864,-179.307,5.249,148.698
C01399=1238.129,6.123,-40.879,-179.305,5.249,148.697
C01400=1238.124,6.372,-40.894,-179.301,5.249,148.696
C01401=1238.119,6.622,-40.909,-179.299,5.249,148.695
C01402=1238.114,6.871,-40.924,-179.297,5.249,148.695
C01403=1238.109,7.121,-40.939,-179.294,5.250,148.694
C01404=1238.104,7.370,-40.953,-179.291,5.250,148.693
C01405=1238.099,7.619,-40.968,-179.289,5.250,148.693
C01406=1238.094,7.869,-40.983,-179.287,5.250,148.692
C01407=1238.089,8.119,-40.999,-179.284,5.251,148.691
C01408=1238.085,8.368,-41.014,-179.281,5.252,148.691
C01409=1238.079,8.618,-41.028,-179.279,5.251,148.690
C01410=1238.074,8.867,-41.043,-179.277,5.252,148.689
C01411=1238.069,9.118,-41.058,-179.274,5.252,148.689
C01412=1238.064,9.367,-41.073,-179.272,5.252,148.688
C01413=1238.059,9.616,-41.088,-179.269,5.253,148.687
C01414=1238.054,9.866,-41.103,-179.267,5.253,148.687
C01415=1238.049,10.115,-41.118,-179.264,5.254,148.686
C01416=1238.044,10.364,-41.134,-179.262,5.253,148.685
C01417=1238.039,10.614,-41.148,-179.259,5.254,148.684
C01418=1238.035,10.864,-41.163,-179.257,5.255,148.684
C01419=1238.029,11.113,-41.179,-179.254,5.254,148.683
C01420=1238.024,11.363,-41.193,-179.252,5.255,148.682
C01421=1238.019,11.612,-41.209,-179.249,5.255,148.682
C01422=1238.014,11.861,-41.224,-179.247,5.256,148.681
C01423=1238.009,12.111,-41.239,-179.244,5.256,148.680
C01424=1238.004,12.360,-41.254,-179.242,5.256,148.680
C01425=1237.999,12.610,-41.269,-179.239,5.256,148.679
C01426=1237.995,12.860,-41.285,-179.237,5.256,148.678
C01427=1237.989,13.110,-41.300,-179.234,5.257,148.677
C01428=1237.984,13.359,-41.315,-179.231,5.257,148.677
C01429=1237.980,13.608,-41.330,-179.229,5.258,148.676
C01430=1237.974,13.857,-41.345,-179.227,5.257,148.675
C01431=1237.970,14.106,-41.360,-179.224,5.258,148.675
C01432=1237.964,14.356,-41.375,-179.221,5.259,148.674
C01433=1237.960,14.606,-41.390,-179.219,5.259,148.673
C01434=1237.954,14.856,-41.406,-179.217,5.259,148.673
C01435=1237.949,15.105,-41.422,-179.214,5.259,148.672
C01436=1237.944,15.354,-41.437,-179.211,5.260,148.671
C01437=1237.939,15.604,-41.451,-179.209,5.260,148.671
C01438=1237.934,15.853,-41.466,-179.207,5.260,148.670
C01439=1237.929,16.103,-41.482,-179.204,5.261,148.669
C01440=1237.925,16.352,-41.497,-179.201,5.261,148.668
C01441=1237.919,16.602,-41.513,-179.199,5.261,148.668
C01442=1237.915,16.851,-41.528,-179.197,5.262,148.667
C01443=1237.909,17.100,-41.544,-179.194,5.262,148.666
C01444=1237.905,17.351,-41.558,-179.191,5.263,148.666
C01445=1237.899,17.600,-41.574,-179.189,5.262,148.665
C01446=1237.894,17.849,-41.589,-179.186,5.263,148.664
C01447=1237.889,18.099,-41.604,-179.184,5.264,148.664
C01448=1237.884,18.348,-41.620,-179.181,5.264,148.663
C01449=1237.880,18.598,-41.635,-179.179,5.264,148.662
C01450=1237.875,18.847,-41.651,-179.176,5.264,148.662
C01451=1237.869,19.097,-41.666,-179.174,5.265,148.661
C01452=1237.865,19.346,-41.681,-179.171,5.266,148.660
C01453=1237.860,19.596,-41.697,-179.169,5.265,148.660
C01454=1237.855,19.845,-41.712,-179.166,5.266,148.659
C01455=1237.850,20.094,-41.728,-179.164,5.266,148.658
C01456=1237.844,20.344,-41.744,-179.161,5.267,148.658
C01457=1237.840,20.593,-41.759,-179.159,5.267,148.657
C01458=1237.835,20.843,-41.774,-179.156,5.267,148.656
C01459=1237.830,21.092,-41.790,-179.154,5.268,148.655
C01460=1237.825,21.341,-41.805,-179.151,5.268,148.655
C01461=1237.820,21.591,-41.821,-179.149,5.268,148.654
C01462=1237.815,21.841,-41.837,-179.146,5.269,148.653
C01463=1237.810,22.090,-41.852,-179.144,5.269,148.653
C01464=1237.805,22.339,-41.867,-179.141,5.270,148.652
C01465=1237.800,22.589,-41.883,-179.139,5.269,148.651
C01466=1237.795,22.839,-41.898,-179.136,5.270,148.651
C01467=1237.790,23.088,-41.914,-179.134,5.271,148.650
C01468=1237.784,23.337,-41.929,-179.131,5.271,148.649
C01469=1237.780,23.587,-41.945,-179.129,5.271,148.649
C01470=1237.775,23.837,-41.960,-179.126,5.271,148.648
C01471=1237.770,24.086,-41.976,-179.124,5.272,148.647
C01472=1237.765,24.336,-41.992,-179.121,5.272,148.646
C01473=1237.760,24.585,-42.007,-179.119,5.272,148.646
C01474=1237.755,24.834,-42.023,-179.116,5.272,148.645
C01475=1237.750,25.084,-42.039,-179.113,5.273,148.644
C01476=1237.746,25.333,-42.054,-179.111,5.274,148.644
C01477=1237.740,25.582,-42.070,-179.109,5.273,148.643
C01478=1237.736,25.833,-42.086,-179.106,5.274,148.642
C01479=1237.730,26.082,-42.101,-179.103,5.274,148.642
C01480=1237.725,26.331,-42.117,-179.101,5.275,148.641
C01481=1237.721,26.581,-42.133,-179.098,5.276,148.640
C01482=1237.716,26.830,-42.148,-179.096,5.275,148.640
C01483=1237.710,27.079,-42.164,-179.093,5.276,148.639
C01484=1237.705,27.329,-42.180,-179.091,5.276,148.638
C01485=1237.701,27.579,-42.195,-179.088,5.277,148.638
C01486=1237.696,27.827,-42.211,-179.086,5.277,148.637
C01487=1237.691,28.077,-42.227,-179.083,5.277,148.636
C01488=1237.686,28.327,-42.243,-179.081,5.278,148.635
C01489=1237.680,28.576,-42.258,-179.078,5.278,148.635
C01490=1237.676,28.825,-42.274,-179.076,5.278,148.634
C01491=1237.671,29.075,-42.290,-179.073,5.279,148.633
C01492=1237.666,29.324,-42.306,-179.071,5.279,148.633
C01493=1237.661,29.593,-42.323,-179.068,5.280,148.632
C01494=1237.655,29.862,-42.340,-179.065,5.280,148.631
C01495=1237.650,30.130,-42.357,-179.063,5.281,148.631
C01496=1237.644,30.399,-42.374,-179.060,5.282,148.630
C01497=1237.639,30.649,-42.390,-179.057,5.282,148.629
C01498=1237.635,30.897,-42.406,-179.055,5.282,148.629
C01499=1237.630,31.147,-42.421,-179.053,5.282,148.628
C01500=1237.625,31.397,-42.437,-179.050,5.283,148.627
C01501=1237.620,31.646,-42.454,-179.047,5.284,148.627
C01502=1237.615,31.896,-42.470,-179.045,5.283,148.626
C01503=1237.609,32.145,-42.485,-179.043,5.284,148.625
C01504=1237.605,32.395,-42.502,-179.040,5.284,148.625
C01505=1237.600,32.644,-42.517,-179.037,5.285,148.624
C01506=1237.595,32.893,-42.534,-179.035,5.286,148.623
C01507=1237.590,33.143,-42.550,-179.033,5.285,148.623
C01508=1237.585,33.392,-42.565,-179.030,5.286,148.622
C01509=1237.581,33.642,-42.581,-179.027,5.286,148.621
C01510=1237.575,33.891,-42.597,-179.025,5.287,148.621
C01511=1237.571,34.140,-42.614,-179.022,5.288,148.620
C01512=1237.565,34.390,-42.629,-179.020,5.287,148.619
C01513=1237.560,34.639,-42.645,-179.017,5.288,148.619
C01514=1237.556,34.889,-42.661,-179.015,5.288,148.618
C01515=1237.550,35.138,-42.677,-179.012,5.289,148.617
C01516=1237.546,35.388,-42.694,-179.009,5.290,148.617
C01517=1237.540,35.637,-42.709,-179.007,5.289,148.616
C01518=1237.536,35.887,-42.726,-179.005,5.290,148.615
C01519=1237.530,36.136,-42.742,-179.002,5.290,148.614
C01520=1237.526,36.385,-42.758,-178.999,5.291,148.614
C01521=1237.521,36.635,-42.774,-178.997,5.292,148.613
C01522=1237.516,36.884,-42.790,-178.994,5.292,148.612
C01523=1237.511,37.134,-42.806,-178.992,5.292,148.612
C01524=1237.506,37.383,-42.823,-178.989,5.292,148.611
C01525=1237.501,37.633,-42.838,-178.987,5.293,148.610
C01526=1237.496,37.882,-42.855,-178.984,5.294,148.610
C01527=1237.491,38.131,-42.871,-178.982,5.294,148.609
C01528=1237.486,38.381,-42.887,-178.979,5.294,148.608
C01529=1237.481,38.630,-42.903,-178.977,5.294,148.608
C01530=1237.477,38.880,-42.919,-178.974,5.295,148.607
C01531=1237.471,39.129,-42.936,-178.972,5.296,148.606
C01532=1237.467,39.379,-42.952,-178.969,5.296,148.606
C01533=1237.462,39.628,-42.968,-178.966,5.297,148.605
C01534=1237.457,39.878,-42.984,-178.964,5.297,148.604
C01535=1237.451,40.127,-43.001,-178.962,5.297,148.604
C01536=1237.447,40.376,-43.018,-178.959,5.298,148.603
C01537=1237.441,40.626,-43.033,-178.957,5.299,148.603
C01538=1237.437,40.875,-43.050,-178.954,5.299,148.602
C01539=1237.431,41.124,-43.065,-178.952,5.299,148.601
C01540=1237.427,41.374,-43.082,-178.949,5.299,148.601
C01541=1237.422,41.623,-43.098,-178.947,5.300,148.600
C01542=1237.417,41.873,-43.114,-178.944,5.301,148.599
C01543=1237.412,42.122,-43.131,-178.941,5.301,148.599
C01544=1237.407,42.371,-43.148,-178.939,5.302,148.598
C01545=1237.402,42.622,-43.164,-178.937,5.302,148.597
C01546=1237.397,42.870,-43.180,-178.934,5.302,148.596
C01547=1237.392,43.120,-43.197,-178.931,5.303,148.596
C01548=1237.387,43.369,-43.213,-178.929,5.303,148.595
C01549=1237.382,43.619,-43.229,-178.926,5.304,148.594
C01550=1237.378,43.868,-43.246,-178.924,5.304,148.594
C01551=1237.372,44.117,-43.263,-178.921,5.304,148.593
C01552=1237.367,44.367,-43.279,-178.919,5.305,148.592
C01553=1237.362,44.616,-43.295,-178.916,5.305,148.592
C01554=1237.358,44.866,-43.312,-178.914,5.306,148.591
C01555=1237.353,45.115,-43.328,-178.911,5.306,148.590
C01556=1237.347,45.364,-43.345,-178.908,5.307,148.590
C01557=1237.343,45.614,-43.361,-178.906,5.308,148.589
C01558=1237.338,45.863,-43.377,-178.904,5.307,148.588
C01559=1237.333,46.113,-43.394,-178.901,5.308,148.588
C01560=1237.329,46.362,-43.411,-178.899,5.309,148.587
C01561=1237.323,46.611,-43.428,-178.896,5.309,148.587
C01562=1237.318,46.861,-43.444,-178.894,5.310,148.586
C01563=1237.314,47.111,-43.460,-178.891,5.311,148.585
C01564=1237.308,47.360,-43.477,-178.888,5.311,148.585
C01565=1237.303,47.609,-43.494,-178.886,5.311,148.584
C01566=1237.298,47.858,-43.510,-178.884,5.312,148.583
C01567=1237.294,48.108,-43.527,-178.881,5.312,148.583
C01568=1237.289,48.358,-43.543,-178.878,5.313,148.582
C01569=1237.283,48.607,-43.560,-178.876,5.313,148.581
C01570=1237.279,48.856,-43.576,-178.873,5.314,148.581
C01571=1237.274,49.106,-43.593,-178.870,5.314,148.580
C01572=1237.269,49.355,-43.609,-178.868,5.314,148.579
C01573=1237.264,49.604,-43.627,-178.866,5.315,148.579
C01574=1237.259,49.854,-43.643,-178.863,5.315,148.578
C01575=1237.254,50.103,-43.660,-178.861,5.316,148.577
C01576=1237.249,50.352,-43.677,-178.858,5.317,148.577
C01577=1237.245,50.602,-43.693,-178.856,5.317,148.576
C01578=1237.240,50.851,-43.710,-178.853,5.318,148.575
C01579=1237.234,51.100,-43.727,-178.851,5.318,148.575
C01580=1237.230,51.350,-43.744,-178.848,5.318,148.574
C01581=1237.225,51.599,-43.760,-178.846,5.319,148.573
C01582=1237.220,51.849,-43.777,-178.843,5.319,148.573
C01583=1237.215,52.098,-43.794,-178.840,5.320,148.572
C01584=1237.211,52.348,-43.811,-178.838,5.321,148.571
C01585=1237.205,52.597,-43.827,-178.835,5.321,148.571
C01586=1237.200,52.846,-43.844,-178.832,5.322,148.570
C01587=1237.196,53.096,-43.861,-178.830,5.322,148.569
C01588=1237.191,53.345,-43.878,-178.828,5.322,148.569
C01589=1237.185,53.594,-43.894,-178.826,5.323,148.568
C01590=1237.181,53.844,-43.911,-178.823,5.324,148.568
C01591=1237.176,54.093,-43.928,-178.820,5.324,148.567
C01592=1237.171,54.343,-43.945,-178.818,5.325,148.566
C01593=1237.165,54.592,-43.962,-178.815,5.325,148.566
C01594=1237.161,54.841,-43.979,-178.812,5.326,148.565
C01595=1237.156,55.091,-43.996,-178.810,5.327,148.564
C01596=1237.151,55.341,-44.013,-178.808,5.326,148.564
C01597=1237.146,55.609,-44.030,-178.805,5.327,148.563
C01598=1237.141,55.878,-44.049,-178.802,5.328,148.562
C01599=1237.135,56.145,-44.067,-178.799,5.329,148.562
C01600=1237.130,56.414,-44.085,-178.797,5.330,148.561
C01601=1237.126,56.664,-44.102,-178.795,5.329,148.560
C01602=1237.120,56.912,-44.120,-178.792,5.330,148.560
C01603=1237.116,57.162,-44.136,-178.789,5.330,148.559
C01604=1237.110,57.411,-44.154,-178.787,5.331,148.558
C01605=1237.106,57.661,-44.170,-178.784,5.332,148.558
C01606=1237.100,57.910,-44.187,-178.781,5.332,148.557
C01607=1237.096,58.160,-44.204,-178.779,5.333,148.556
C01608=1237.091,58.409,-44.222,-178.776,5.333,148.556
C01609=1237.086,58.658,-44.238,-178.773,5.334,148.555
C01610=1237.081,58.908,-44.256,-178.771,5.335,148.554
C01611=1237.076,59.157,-44.272,-178.769,5.335,148.554
C01612=1237.071,59.406,-44.290,-178.767,5.335,148.553
C01613=1237.066,59.655,-44.307,-178.764,5.336,148.552
C01614=1237.061,59.905,-44.324,-178.761,5.336,148.552
C01615=1237.057,60.155,-44.341,-178.759,5.337,148.551
C01616=1237.052,60.404,-44.359,-178.756,5.338,148.550
C01617=1237.046,60.653,-44.375,-178.753,5.338,148.550
C01618=1237.042,60.902,-44.392,-178.751,5.339,148.549
C01619=1237.036,61.152,-44.409,-178.748,5.339,148.548
C01620=1237.032,61.401,-44.427,-178.746,5.340,148.548
C01621=1237.027,61.651,-44.444,-178.743,5.341,148.547
C01622=1237.022,61.900,-44.461,-178.741,5.341,148.547
C01623=1237.018,62.150,-44.479,-178.739,5.341,148.546
C01624=1237.012,62.399,-44.496,-178.736,5.342,148.545
C01625=1237.007,62.648,-44.512,-178.733,5.342,148.545
C01626=1237.002,62.897,-44.530,-178.731,5.343,148.544
C01627=1236.998,63.147,-44.547,-178.728,5.344,148.543
C01628=1236.993,63.396,-44.565,-178.726,5.344,148.543
C01629=1236.988,63.646,-44.582,-178.723,5.345,148.542
C01630=1236.983,63.895,-44.599,-178.721,5.346,148.542
C01631=1236.978,64.144,-44.617,-178.718,5.346,148.541
C01632=1236.973,64.393,-44.633,-178.716,5.347,148.540
C01633=1236.968,64.642,-44.651,-178.713,5.348,148.540
C01634=1236.963,64.892,-44.668,-178.710,5.348,148.539
C01635=1236.959,65.142,-44.685,-178.708,5.349,148.538
C01636=1236.954,65.391,-44.703,-178.706,5.348,148.538
C01637=1236.949,65.641,-44.720,-178.703,5.349,148.537
C01638=1236.944,65.890,-44.738,-178.701,5.350,148.537
C01639=1236.939,66.139,-44.755,-178.698,5.351,148.536
C01640=1236.934,66.388,-44.773,-178.696,5.351,148.535
C01641=1236.930,66.638,-44.790,-178.693,5.352,148.535
C01642=1236.925,66.887,-44.808,-178.690,5.352,148.534
C01643=1236.919,67.136,-44.824,-178.688,5.353,148.533
C01644=1236.915,67.385,-44.842,-178.685,5.354,148.533
C01645=1236.910,67.635,-44.859,-178.683,5.355,148.532
C01646=1236.905,67.884,-44.877,-178.680,5.355,148.531
C01647=1236.899,68.134,-44.894,-178.678,5.356,148.531
C01648=1236.895,68.383,-44.912,-178.675,5.356,148.530
C01649=1236.890,68.633,-44.929,-178.672,5.357,148.529
C01650=1236.885,68.882,-44.947,-178.670,5.357,148.529
C01651=1236.880,69.132,-44.964,-178.667,5.358,148.528
C01652=1236.876,69.380,-44.982,-178.665,5.359,148.528
C01653=1236.871,69.630,-45.000,-178.663,5.359,148.527
C01654=1236.866,69.879,-45.017,-178.660,5.359,148.526
C01655=1236.861,70.129,-45.035,-178.658,5.360,148.526
C01656=1236.856,70.378,-45.052,-178.655,5.361,148.525
C01657=1236.851,70.627,-45.070,-178.652,5.361,148.524
C01658=1236.846,70.876,-45.087,-178.650,5.362,148.524
C01659=1236.841,71.126,-45.105,-178.648,5.363,148.523
C01660=1236.837,71.375,-45.122,-178.645,5.363,148.523
C01661=1236.832,71.624,-45.140,-178.642,5.364,148.522
C01662=1236.827,71.874,-45.157,-178.640,5.365,148.521
C01663=1236.822,72.123,-45.175,-178.637,5.365,148.521
C01664=1236.817,72.372,-45.193,-178.635,5.366,148.520
C01665=1236.812,72.622,-45.211,-178.632,5.366,148.519
C01666=1236.808,72.871,-45.228,-178.630,5.367,148.519
C01667=1236.803,73.120,-45.246,-178.627,5.368,148.518
C01668=1236.798,73.370,-45.263,-178.624,5.368,148.518
C01669=1236.793,73.619,-45.281,-178.622,5.369,148.517
C01670=1236.788,73.868,-45.299,-178.619,5.370,148.516
C01671=1236.783,74.118,-45.316,-178.617,5.370,148.516
C01672=1236.778,74.367,-45.334,-178.614,5.371,148.515
C01673=1236.773,74.616,-45.352,-178.612,5.372,148.515
C01674=1236.769,74.865,-45.370,-178.609,5.372,148.514
C01675=1236.763,75.115,-45.387,-178.607,5.373,148.513
C01676=1236.758,75.364,-45.405,-178.604,5.374,148.513
C01677=1236.753,75.613,-45.423,-178.601,5.374,148.512
C01678=1236.749,75.863,-45.441,-178.599,5.375,148.511
C01679=1236.744,76.113,-45.459,-178.597,5.376,148.511
C01680=1236.739,76.362,-45.477,-178.594,5.376,148.510
C01681=1236.734,76.612,-45.495,-178.591,5.377,148.509
C01682=1236.730,76.860,-45.512,-178.589,5.378,148.509
C01683=1236.725,77.110,-45.530,-178.586,5.378,148.508
C01684=1236.720,77.359,-45.548,-178.583,5.379,148.508
C01685=1236.715,77.608,-45.566,-178.581,5.380,148.507
C01686=1236.710,77.858,-45.583,-178.579,5.380,148.506
C01687=1236.705,78.107,-45.601,-178.576,5.381,148.506
C01688=1236.700,78.356,-45.619,-178.573,5.382,148.505
C01689=1236.695,78.605,-45.637,-178.571,5.382,148.504
C01690=1236.691,78.855,-45.655,-178.569,5.383,148.504
C01691=1236.686,79.104,-45.673,-178.566,5.384,148.503
C01692=1236.681,79.353,-45.691,-178.563,5.384,148.503
C01693=1236.676,79.603,-45.709,-178.561,5.385,148.502
C01694=1236.671,79.852,-45.727,-178.558,5.386,148.501
C01695=1236.666,80.101,-45.745,-178.556,5.386,148.501
C01696=1236.661,80.350,-45.763,-178.553,5.387,148.500
C01697=1236.657,80.599,-45.781,-178.551,5.388,148.500
C01698=1236.652,80.850,-45.799,-178.548,5.388,148.499
C01699=1236.647,81.099,-45.817,-178.546,5.389,148.498
C01700=1236.642,81.348,-45.835,-178.543,5.390,148.498
C01701=1236.637,81.616,-45.854,-178.540,5.390,148.497
C01702=1236.631,81.885,-45.874,-178.538,5.391,148.496
C01703=1236.626,82.153,-45.894,-178.535,5.391,148.496
C01704=1236.621,82.421,-45.913,-178.532,5.392,148.495
C01705=1236.616,82.671,-45.931,-178.530,5.393,148.494
C01706=1236.611,82.920,-45.949,-178.528,5.393,148.494
C01707=1236.606,83.169,-45.967,-178.525,5.394,148.493
C01708=1236.602,83.419,-45.985,-178.522,5.395,148.493
C01709=1236.597,83.668,-46.003,-178.520,5.395,148.492
C01710=1236.592,83.917,-46.021,-178.517,5.396,148.491
C01711=1236.587,84.166,-46.039,-178.515,5.397,148.491
C01712=1236.582,84.416,-46.058,-178.512,5.397,148.490
C01713=1236.578,84.665,-46.077,-178.510,5.398,148.490
C01714=1236.573,84.914,-46.095,-178.507,5.399,148.489
C01715=1236.568,85.164,-46.113,-178.505,5.399,148.488
C01716=1236.563,85.413,-46.131,-178.502,5.400,148.488
C01717=1236.558,85.662,-46.149,-178.500,5.401,148.487
C01718=1236.554,85.912,-46.167,-178.497,5.402,148.487
C01719=1236.549,86.161,-46.185,-178.494,5.403,148.486
C01720=1236.543,86.410,-46.204,-178.491,5.404,148.485
C01721=1236.539,86.659,-46.223,-178.489,5.404,148.485
C01722=1236.534,86.908,-46.241,-178.487,5.405,148.484
C01723=1236.529,87.158,-46.259,-178.484,5.406,148.484
C01724=1236.524,87.407,-46.277,-178.481,5.406,148.483
C01725=1236.519,87.656,-46.295,-178.479,5.407,148.482
C01726=1236.514,87.905,-46.314,-178.477,5.408,148.482
C01727=1236.510,88.155,-46.332,-178.474,5.409,148.481
C01728=1236.505,88.404,-46.350,-178.471,5.409,148.481
C01729=1236.500,88.653,-46.368,-178.469,5.410,148.480
C01730=1236.495,88.903,-46.386,-178.467,5.411,148.479
C01731=1236.490,89.152,-46.406,-178.464,5.411,148.479
C01732=1236.485,89.401,-46.424,-178.461,5.412,148.478
C01733=1236.480,89.651,-46.442,-178.459,5.413,148.477
C01734=1236.476,89.900,-46.461,-178.456,5.413,148.477
C01735=1236.471,90.149,-46.480,-178.454,5.414,148.476
C01736=1236.466,90.398,-46.498,-178.451,5.415,148.476
C01737=1236.461,90.648,-46.516,-178.449,5.415,148.475
C01738=1236.457,90.897,-46.535,-178.446,5.416,148.474
C01739=1236.451,91.146,-46.553,-178.444,5.417,148.474
C01740=1236.446,91.396,-46.571,-178.441,5.418,148.473
C01741=1236.442,91.645,-46.590,-178.438,5.419,148.473
C01742=1236.437,91.894,-46.609,-178.436,5.420,148.472
C01743=1236.432,92.143,-46.627,-178.433,5.421,148.472
C01744=1236.428,92.393,-46.646,-178.431,5.421,148.471
C01745=1236.423,92.642,-46.664,-178.428,5.422,148.470
C01746=1236.418,92.891,-46.683,-178.426,5.422,148.470
C01747=1236.413,93.140,-46.701,-178.423,5.423,148.469
C01748=1236.408,93.390,-46.719,-178.421,5.424,148.469
C01749=1236.403,93.639,-46.739,-178.418,5.425,148.468
C01750=1236.399,93.889,-46.757,-178.416,5.425,148.467
C01751=1236.394,94.137,-46.776,-178.413,5.426,148.467
C01752=1236.388,94.387,-46.794,-178.411,5.427,148.466
C01753=1236.384,94.637,-46.813,-178.408,5.427,148.466
C01754=1236.380,94.885,-46.831,-178.406,5.428,148.465
C01755=1236.374,95.135,-46.850,-178.402,5.429,148.464
C01756=1236.370,95.384,-46.869,-178.400,5.430,148.464
C01757=1236.364,95.633,-46.888,-178.398,5.431,148.463
C01758=1236.360,95.882,-46.906,-178.395,5.432,148.463
C01759=1236.355,96.132,-46.925,-178.392,5.432,148.462
C01760=1236.350,96.381,-46.944,-178.390,5.433,148.462
C01761=1236.345,96.630,-46.962,-178.388,5.434,148.461
C01762=1236.341,96.879,-46.981,-178.385,5.434,148.460
C01763=1236.335,97.129,-47.000,-178.382,5.435,148.460
C01764=1236.331,97.378,-47.019,-178.380,5.436,148.459
C01765=1236.326,97.627,-47.037,-178.378,5.437,148.458
C01766=1236.321,97.876,-47.056,-178.375,5.437,148.458
C01767=1236.316,98.126,-47.075,-178.372,5.439,148.457
C01768=1236.312,98.375,-47.094,-178.370,5.440,148.457
C01769=1236.307,98.624,-47.113,-178.367,5.440,148.456
C01770=1236.302,98.873,-47.131,-178.365,5.441,148.455
C01771=1236.297,99.122,-47.150,-178.362,5.442,148.455
C01772=1236.292,99.372,-47.169,-178.360,5.443,148.454
C01773=1236.288,99.621,-47.188,-178.357,5.443,148.454
C01774=1236.283,99.870,-47.207,-178.355,5.444,148.453
C01775=1236.278,100.119,-47.225,-178.352,5.445,148.453
C01776=1236.273,100.369,-47.245,-178.350,5.445,148.452
C01777=1236.269,100.617,-47.264,-178.347,5.446,148.451
C01778=1236.264,100.868,-47.282,-178.344,5.447,148.451
C01779=1236.259,101.116,-47.301,-178.342,5.448,148.450
C01780=1236.254,101.365,-47.320,-178.339,5.449,148.450
C01781=1236.249,101.615,-47.339,-178.337,5.450,148.449
C01782=1236.244,101.864,-47.358,-178.335,5.451,148.449
C01783=1236.240,102.113,-47.377,-178.332,5.451,148.448
C01784=1236.234,102.363,-47.396,-178.329,5.452,148.447
C01785=1236.230,102.612,-47.415,-178.327,5.452,148.447
C01786=1236.225,102.861,-47.434,-178.325,5.453,148.446
C01787=1236.220,103.110,-47.454,-178.321,5.455,148.446
C01788=1236.215,103.359,-47.472,-178.319,5.455,148.445
C01789=1236.211,103.609,-47.491,-178.317,5.456,148.445
C01790=1236.206,103.858,-47.510,-178.314,5.457,148.444
C01791=1236.201,104.107,-47.530,-178.311,5.458,148.443
C01792=1236.196,104.357,-47.548,-178.309,5.458,148.443
C01793=1236.192,104.606,-47.567,-178.307,5.459,148.442
C01794=1236.186,104.855,-47.587,-178.304,5.460,148.442
C01795=1236.182,105.104,-47.606,-178.301,5.461,148.441
C01796=1236.177,105.353,-47.625,-178.299,5.462,148.441
C01797=1236.172,105.603,-47.644,-178.296,5.463,148.440
C01798=1236.167,105.852,-47.663,-178.294,5.464,148.439
C01799=1236.162,106.101,-47.682,-178.291,5.465,148.439
C01800=1236.158,106.350,-47.701,-178.289,5.465,148.438
C01801=1236.153,106.599,-47.721,-178.286,5.466,148.438
C01802=1236.148,106.848,-47.740,-178.283,5.467,148.437
C01803=1236.144,107.097,-47.759,-178.281,5.468,148.437
C01804=1236.139,107.348,-47.778,-178.278,5.469,148.436
C01805=1236.133,107.616,-47.799,-178.276,5.470,148.435
C01806=1236.128,107.884,-47.820,-178.273,5.470,148.435
C01807=1236.123,108.152,-47.840,-178.270,5.472,148.434
C01808=1236.118,108.421,-47.862,-178.267,5.472,148.433
C01809=1236.113,108.669,-47.880,-178.265,5.473,148.433
C01810=1236.108,108.920,-47.899,-178.263,5.474,148.432
C01811=1236.103,109.169,-47.919,-178.260,5.474,148.432
C01812=1236.098,109.418,-47.938,-178.257,5.476,148.431
C01813=1236.094,109.667,-47.957,-178.255,5.477,148.431
C01814=1236.089,109.916,-47.976,-178.252,5.478,148.430
C01815=1236.084,110.166,-47.996,-178.250,5.478,148.430
C01816=1236.080,110.415,-48.015,-178.247,5.479,148.429
C01817=1236.075,110.664,-48.034,-178.245,5.480,148.428
C01818=1236.070,110.913,-48.054,-178.242,5.482,148.428
C01819=1236.065,111.162,-48.073,-178.239,5.482,148.427
C01820=1236.061,111.412,-48.092,-178.237,5.483,148.427
C01821=1236.056,111.661,-48.112,-178.235,5.484,148.426
C01822=1236.051,111.909,-48.132,-178.232,5.484,148.425
C01823=1236.046,112.159,-48.152,-178.229,5.485,148.425
C01824=1236.041,112.408,-48.171,-178.227,5.487,148.424
C01825=1236.037,112.657,-48.190,-178.224,5.487,148.424
C01826=1236.032,112.907,-48.210,-178.222,5.488,148.423
C01827=1236.027,113.155,-48.229,-178.219,5.489,148.423
C01828=1236.022,113.405,-48.249,-178.217,5.490,148.422
C01829=1236.017,113.655,-48.268,-178.214,5.490,148.421
C01830=1236.013,113.903,-48.287,-178.212,5.492,148.421
C01831=1236.008,114.153,-48.307,-178.209,5.493,148.420
